	{attribute 'TcIecLibraryType'}
	{attribute 'external_name' := 'F_VN_BrightBorderObjects_GUID_85963068_12EB_DB9B_82A7_C723E1DC205C'}
	(* Find bright objects connected to the image border within a gray-scale single-channel image. *)
	FUNCTION F_VN_BrightBorderObjects : HRESULT
	VAR_INPUT
		ipSrcImage	:	ITcVnImage;	(* Source image (USINT, UINT, INT, REAL, or LREAL, 1 channel) *)
		ipDestImage	:	REFERENCE TO ITcVnImage;	(* Destination image (An appropriate destination image will be created if required.) *)
		hrPrev	:	HRESULT;	(* HRESULT indicating the result of previous operations (If SUCCEEDED(hrPrev) equals false, no operation is executed.) *)
	END_VAR

END_FUNCTION

// Functions/Image Filtering/F_VN_CreateStructuringElement

	{attribute 'TcIecLibraryType'}
	{attribute 'external_name' := 'F_VN_CreateStructuringElement_GUID_A74CE5A4_39AA_D057_BA78_297FA60F12C8'}
	(* Creates a structuring element for the usage with morphological operators and allocate an appropriate data buffer. The initial reference count is set to one if a new image interface is created and kept, otherwise. *)
	FUNCTION F_VN_CreateStructuringElement : HRESULT
	VAR_INPUT
		ipStructuringElement	:	REFERENCE TO ITcVnImage;	(* Returns the created structuring element (Non-zero interface pointers are reused.) *)
		eShape	:	ETcVnStructuringElementShape;	(* Shape of the structuring element (rectangle, cross, or ellipse) *)
		nWidth	:	UDINT;	(* Width *)
		nHeight	:	UDINT;	(* Height *)
		hrPrev	:	HRESULT;	(* HRESULT indicating the result of previous operations (If SUCCEEDED(hrPrev) equals false, no operation is executed.) *)
	END_VAR

END_FUNCTION

// Functions/Image Filtering/F_VN_CustomFilter

	{attribute 'TcIecLibraryType'}
	{attribute 'external_name' := 'F_VN_CustomFilter_GUID_4301F747_474B_D00C_9989_9E35727DC697'}
	(* Apply a custom filter to the image. *)
	FUNCTION F_VN_CustomFilter : HRESULT
	VAR_INPUT
		ipSrcImage	:	ITcVnImage;	(* Source image *)
		ipDestImage	:	REFERENCE TO ITcVnImage;	(* Destination image (An appropriate destination image will be created if required.) *)
		eDestDepth	:	ETcVnElementType;	(* Destination image depth *)
	END_VAR
	VAR_IN_OUT
		stKernel	:	TcVnMatrix;	(* Custom filter kernel with values of type REAL or LREAL *)
	END_VAR
	VAR_INPUT
		hrPrev	:	HRESULT;	(* HRESULT indicating the result of previous operations (If SUCCEEDED(hrPrev) equals false, no operation is executed.) *)
	END_VAR

END_FUNCTION

// Functions/Image Filtering/F_VN_CustomFilterExp

	{attribute 'TcIecLibraryType'}
	{attribute 'external_name' := 'F_VN_CustomFilterExp_GUID_6B16FEA9_6021_D269_AEDC_2F022CED5005'}
	(* Apply a custom filter to the image. (expert function) *)
	FUNCTION F_VN_CustomFilterExp : HRESULT
	VAR_INPUT
		ipSrcImage	:	ITcVnImage;	(* Source image *)
		ipDestImage	:	REFERENCE TO ITcVnImage;	(* Destination image (An appropriate destination image will be created if required.) *)
		eDestDepth	:	ETcVnElementType;	(* Destination image depth *)
	END_VAR
	VAR_IN_OUT
		stKernel	:	TcVnMatrix;	(* Custom filter kernel with values of type REAL or LREAL *)
		aAnchor	:	TcVnPoint;	(* Anchor point of the kernel *)
	END_VAR
	VAR_INPUT
		fDelta	:	LREAL;	(* Value added to each pixel after filtering *)
		eBorderType	:	ETcVnBorderInterpolationMethod;	(* Image border handling *)
		hrPrev	:	HRESULT;	(* HRESULT indicating the result of previous operations (If SUCCEEDED(hrPrev) equals false, no operation is executed.) *)
	END_VAR

END_FUNCTION

// Functions/Image Filtering/F_VN_DarkBorderObjects

	{attribute 'TcIecLibraryType'}
	{attribute 'external_name' := 'F_VN_DarkBorderObjects_GUID_502A5401_CBE1_DB60_8EE9_DC582F5D3E12'}
	(* Find dark objects connected to the image border within a gray-scale single-channel image. (equivalent to filling holes) *)
	FUNCTION F_VN_DarkBorderObjects : HRESULT
	VAR_INPUT
		ipSrcImage	:	ITcVnImage;	(* Source image (USINT, UINT, INT, REAL, or LREAL, 1 channel) *)
		ipDestImage	:	REFERENCE TO ITcVnImage;	(* Destination image (An appropriate destination image will be created if required.) *)
		hrPrev	:	HRESULT;	(* HRESULT indicating the result of previous operations (If SUCCEEDED(hrPrev) equals false, no operation is executed.) *)
	END_VAR

END_FUNCTION

// Functions/Image Filtering/F_VN_FillHoles

	{attribute 'TcIecLibraryType'}
	{attribute 'external_name' := 'F_VN_FillHoles_GUID_355DF251_1290_D7ED_B630_2E4E8A66643C'}
	(* Fill holes within a gray-scale single-channel image. (equivalent to finding dark border objects) *)
	FUNCTION F_VN_FillHoles : HRESULT
	VAR_INPUT
		ipSrcImage	:	ITcVnImage;	(* Source image (USINT, UINT, INT, REAL, or LREAL, 1 channel) *)
		ipDestImage	:	REFERENCE TO ITcVnImage;	(* Destination image (An appropriate destination image will be created if required.) *)
		hrPrev	:	HRESULT;	(* HRESULT indicating the result of previous operations (If SUCCEEDED(hrPrev) equals false, no operation is executed.) *)
	END_VAR

END_FUNCTION

// Functions/Image Filtering/F_VN_GaussianFilter

	{attribute 'TcIecLibraryType'}
	{attribute 'external_name' := 'F_VN_GaussianFilter_GUID_E5394B01_3A0E_DAE0_9B18_9A4594D869A5'}
	(* Apply a Gaussian filter to smooth the image. *)
	FUNCTION F_VN_GaussianFilter : HRESULT
	VAR_INPUT
		ipSrcImage	:	ITcVnImage;	(* Source image *)
		ipDestImage	:	REFERENCE TO ITcVnImage;	(* Destination image (An appropriate destination image will be created if required.) *)
		nFilterWidth	:	UDINT;	(* Filter width in pixels (1, 3, 5, 7, ...) *)
		nFilterHeight	:	UDINT;	(* Filter height in pixels (1, 3, 5, 7, ...) *)
		hrPrev	:	HRESULT;	(* HRESULT indicating the result of previous operations (If SUCCEEDED(hrPrev) equals false, no operation is executed.) *)
	END_VAR

END_FUNCTION

// Functions/Image Filtering/F_VN_GaussianFilterExp

	{attribute 'TcIecLibraryType'}
	{attribute 'external_name' := 'F_VN_GaussianFilterExp_GUID_34305DF4_4689_DEA9_9855_ED8AC64FC35B'}
	(* Apply a Gaussian filter to smooth the image. (expert function) *)
	FUNCTION F_VN_GaussianFilterExp : HRESULT
	VAR_INPUT
		ipSrcImage	:	ITcVnImage;	(* Source image *)
		ipDestImage	:	REFERENCE TO ITcVnImage;	(* Destination image (An appropriate destination image will be created if required.) *)
		nFilterWidth	:	UDINT;	(* Filter width in pixels (1, 3, 5, 7, ...) *)
		nFilterHeight	:	UDINT;	(* Filter height in pixels (1, 3, 5, 7, ...) *)
		fSigmaX	:	LREAL;	(* Gaussian kernel standard deviation in X direction (>= 0, automatically chosen if 0) *)
		fSigmaY	:	LREAL;	(* Gaussian kernel standard deviation in Y direction (>= 0, automatically chosen if 0) *)
		eBorderType	:	ETcVnBorderInterpolationMethod;	(* Image border handling *)
		hrPrev	:	HRESULT;	(* HRESULT indicating the result of previous operations (If SUCCEEDED(hrPrev) equals false, no operation is executed.) *)
	END_VAR

END_FUNCTION

// Functions/Image Filtering/F_VN_LaplacianFilter

	{attribute 'TcIecLibraryType'}
	{attribute 'external_name' := 'F_VN_LaplacianFilter_GUID_52689B07_71D3_DE56_A0C0_525AA2EFFA66'}
	(* Apply a Laplacian filter to an image. *)
	FUNCTION F_VN_LaplacianFilter : HRESULT
	VAR_INPUT
		ipSrcImage	:	ITcVnImage;	(* Source image *)
		ipDestImage	:	REFERENCE TO ITcVnImage;	(* Destination image (An appropriate destination image will be created if required.) *)
		eDestDepth	:	ETcVnElementType;	(* Destination image depth *)
		hrPrev	:	HRESULT;	(* HRESULT indicating the result of previous operations (If SUCCEEDED(hrPrev) equals false, no operation is executed.) *)
	END_VAR

END_FUNCTION

// Functions/Image Filtering/F_VN_LaplacianFilterExp

	{attribute 'TcIecLibraryType'}
	{attribute 'external_name' := 'F_VN_LaplacianFilterExp_GUID_F05E54BA_3338_DB0A_A7D6_DE17DEB649CB'}
	(* Apply a Laplacian filter to an image. (expert function) *)
	FUNCTION F_VN_LaplacianFilterExp : HRESULT
	VAR_INPUT
		ipSrcImage	:	ITcVnImage;	(* Source image *)
		ipDestImage	:	REFERENCE TO ITcVnImage;	(* Destination image (An appropriate destination image will be created if required.) *)
		eDestDepth	:	ETcVnElementType;	(* Destination image depth *)
		nKernelSize	:	UDINT;	(* Aperture size used to compute the second-derivative filters (1, 3, 5, ..., 31) *)
		fScale	:	LREAL;	(* Scale factor for the computed derivative values *)
		fDelta	:	LREAL;	(* Delta value that is added to the results before storing them *)
		eBorderType	:	ETcVnBorderInterpolationMethod;	(* Image border handling *)
		hrPrev	:	HRESULT;	(* HRESULT indicating the result of previous operations (If SUCCEEDED(hrPrev) equals false, no operation is executed.) *)
	END_VAR

END_FUNCTION

// Functions/Image Filtering/F_VN_LocalMaxima

	{attribute 'TcIecLibraryType'}
	{attribute 'external_name' := 'F_VN_LocalMaxima_GUID_73E2BFA3_7B8C_D368_9D3A_ABFF9FB011DB'}
	(* Find local maxima in a gray-scale single-channel image. The found maxima are marked by a value of 1 in the destination image. *)
	FUNCTION F_VN_LocalMaxima : HRESULT
	VAR_INPUT
		ipSrcImage	:	ITcVnImage;	(* Source image (USINT or UINT, 1 channel) *)
		ipDestImage	:	REFERENCE TO ITcVnImage;	(* Destination image (Must be different from ipSrcImage! An appropriate destination image will be created if required.) *)
		hrPrev	:	HRESULT;	(* HRESULT indicating the result of previous operations (If SUCCEEDED(hrPrev) equals false, no operation is executed.) *)
	END_VAR

END_FUNCTION

// Functions/Image Filtering/F_VN_LocalMinima

	{attribute 'TcIecLibraryType'}
	{attribute 'external_name' := 'F_VN_LocalMinima_GUID_43B2D13E_E00E_D8F8_8DF7_26EA4EF5D134'}
	(* Find local minima in a gray-scale single-channel image. The found minima are marked by a value of 1 in the destination image. *)
	FUNCTION F_VN_LocalMinima : HRESULT
	VAR_INPUT
		ipSrcImage	:	ITcVnImage;	(* Source image (USINT or UINT, 1 channel) *)
		ipDestImage	:	REFERENCE TO ITcVnImage;	(* Destination image (Must be different from ipSrcImage! An appropriate destination image will be created if required.) *)
		hrPrev	:	HRESULT;	(* HRESULT indicating the result of previous operations (If SUCCEEDED(hrPrev) equals false, no operation is executed.) *)
	END_VAR

END_FUNCTION

// Functions/Image Filtering/F_VN_MedianFilter

	{attribute 'TcIecLibraryType'}
	{attribute 'external_name' := 'F_VN_MedianFilter_GUID_68A1C045_786D_D318_9650_B93B817DB87C'}
	(* Apply a Median filter to an image. *)
	FUNCTION F_VN_MedianFilter : HRESULT
	VAR_INPUT
		ipSrcImage	:	ITcVnImage;	(* Source image (for nFilterSize 3 or 5: USINT, UINT, REAL. For bigger filters, only USINT is supported. *)
		ipDestImage	:	REFERENCE TO ITcVnImage;	(* Destination image (An appropriate destination image will be created if required.) *)
		nFilterSize	:	UDINT;	(* Size (width and height) of the filter (3, 5, 7, ...) *)
		hrPrev	:	HRESULT;	(* HRESULT indicating the result of previous operations (If SUCCEEDED(hrPrev) equals false, no operation is executed.) *)
	END_VAR

END_FUNCTION

// Functions/Image Filtering/F_VN_MorphologicalOperator

	{attribute 'TcIecLibraryType'}
	{attribute 'external_name' := 'F_VN_MorphologicalOperator_GUID_C2AADC35_1A3C_DECA_BADD_187CC41E0AFB'}
	(* Apply a morphological operator. *)
	FUNCTION F_VN_MorphologicalOperator : HRESULT
	VAR_INPUT
		ipSrcImage	:	ITcVnImage;	(* Source image (only 1 channel supported for reconstruction operators) *)
		ipDestImage	:	REFERENCE TO ITcVnImage;	(* Destination image (An appropriate destination image will be created if required.) *)
		eOperator	:	ETcVnMorphologicalOperator;	(* Operator type *)
		ipStructuringElement	:	ITcVnImage;	(* Structuring element to be applied (Typically created via F_VN_CreateStructuringElement.) *)
		hrPrev	:	HRESULT;	(* HRESULT indicating the result of previous operations (If SUCCEEDED(hrPrev) equals false, no operation is executed.) *)
	END_VAR

END_FUNCTION

// Functions/Image Filtering/F_VN_RemoveLocalMaxima

	{attribute 'TcIecLibraryType'}
	{attribute 'external_name' := 'F_VN_RemoveLocalMaxima_GUID_133B4553_4F99_DBCD_BA62_EA37E8765D5B'}
	(* Remove local maxima up to a given height from a gray-scale single-channel image. *)
	FUNCTION F_VN_RemoveLocalMaxima : HRESULT
	VAR_INPUT
		ipSrcImage	:	ITcVnImage;	(* Source image (USINT, UINT, INT, REAL, or LREAL, 1 channel) *)
		ipDestImage	:	REFERENCE TO ITcVnImage;	(* Destination image (An appropriate destination image will be created if required.) *)
		fHeight	:	LREAL;	(* Maximum height of the maxima to be removed (must be greater than 0) *)
		hrPrev	:	HRESULT;	(* HRESULT indicating the result of previous operations (If SUCCEEDED(hrPrev) equals false, no operation is executed.) *)
	END_VAR

END_FUNCTION

// Functions/Image Filtering/F_VN_RemoveLocalMinima

	{attribute 'TcIecLibraryType'}
	{attribute 'external_name' := 'F_VN_RemoveLocalMinima_GUID_A59442F0_2AE9_D045_8F9C_09A3C82C0A3B'}
	(* Remove local minima up to a given height from a gray-scale single-channel image. *)
	FUNCTION F_VN_RemoveLocalMinima : HRESULT
	VAR_INPUT
		ipSrcImage	:	ITcVnImage;	(* Source image (USINT, UINT, INT, REAL, or LREAL, 1 channel) *)
		ipDestImage	:	REFERENCE TO ITcVnImage;	(* Destination image (An appropriate destination image will be created if required.) *)
		fHeight	:	LREAL;	(* Maximum height of the minima to be removed (must be greater than 0) *)
		hrPrev	:	HRESULT;	(* HRESULT indicating the result of previous operations (If SUCCEEDED(hrPrev) equals false, no operation is executed.) *)
	END_VAR

END_FUNCTION

// Functions/Image Filtering/F_VN_ScharrFilter

	{attribute 'TcIecLibraryType'}
	{attribute 'external_name' := 'F_VN_ScharrFilter_GUID_3CD4A752_576C_D682_949F_3ED3E34C66A7'}
	(* Calculates the first order derivative in x or y direction using a Scharr filter. *)
	FUNCTION F_VN_ScharrFilter : HRESULT
	VAR_INPUT
		ipSrcImage	:	ITcVnImage;	(* Source image *)
		ipDestImage	:	REFERENCE TO ITcVnImage;	(* Destination image (An appropriate destination image will be created if required.) *)
		eDestDepth	:	ETcVnElementType;	(* Destination image depth *)
		eFilterDirection	:	ETcVnFilterDirection;	(* Filter direction *)
		hrPrev	:	HRESULT;	(* HRESULT indicating the result of previous operations (If SUCCEEDED(hrPrev) equals false, no operation is executed.) *)
	END_VAR

END_FUNCTION

// Functions/Image Filtering/F_VN_ScharrFilterExp

	{attribute 'TcIecLibraryType'}
	{attribute 'external_name' := 'F_VN_ScharrFilterExp_GUID_14964554_311A_DD6B_9094_26927304E48F'}
	(* Calculates the first order derivative in x or y direction using a Scharr filter. (expert function) *)
	FUNCTION F_VN_ScharrFilterExp : HRESULT
	VAR_INPUT
		ipSrcImage	:	ITcVnImage;	(* Source image *)
		ipDestImage	:	REFERENCE TO ITcVnImage;	(* Destination image (An appropriate destination image will be created if required.) *)
		eDestDepth	:	ETcVnElementType;	(* Destination image depth *)
		eFilterDirection	:	ETcVnFilterDirection;	(* Filter direction *)
		fScale	:	LREAL;	(* Scale factor for the computed derivative values *)
		fDelta	:	LREAL;	(* Delta value that is added to the results prior to storing them in dest *)
		eBorderType	:	ETcVnBorderInterpolationMethod;	(* Image border handling *)
		hrPrev	:	HRESULT;	(* HRESULT indicating the result of previous operations (If SUCCEEDED(hrPrev) equals false, no operation is executed.) *)
	END_VAR

END_FUNCTION

// Functions/Image Filtering/F_VN_SeparableCustomFilter

	{attribute 'TcIecLibraryType'}
	{attribute 'external_name' := 'F_VN_SeparableCustomFilter_GUID_638E373F_2CCD_D425_B656_29701E8F04DD'}
	(* Apply a separable custom filter to the image. *)
	FUNCTION F_VN_SeparableCustomFilter : HRESULT
	VAR_INPUT
		ipSrcImage	:	ITcVnImage;	(* Source image *)
		ipDestImage	:	REFERENCE TO ITcVnImage;	(* Destination image (An appropriate destination image will be created if required.) *)
		eDestDepth	:	ETcVnElementType;	(* Destination image depth *)
	END_VAR
	VAR_IN_OUT
		stKernelX	:	TcVnMatrix;	(* 1D custom row-filter kernel with values of type REAL or LREAL *)
		stKernelY	:	TcVnMatrix;	(* 1D custom column-filter kernel with values of type REAL or LREAL *)
	END_VAR
	VAR_INPUT
		hrPrev	:	HRESULT;	(* HRESULT indicating the result of previous operations (If SUCCEEDED(hrPrev) equals false, no operation is executed.) *)
	END_VAR

END_FUNCTION

// Functions/Image Filtering/F_VN_SeparableCustomFilterExp

	{attribute 'TcIecLibraryType'}
	{attribute 'external_name' := 'F_VN_SeparableCustomFilterExp_GUID_CC5A19A5_2D1C_D6B1_9D4E_5D5FBFBA8823'}
	(* Apply a separable custom filter to the image. (expert function) *)
	FUNCTION F_VN_SeparableCustomFilterExp : HRESULT
	VAR_INPUT
		ipSrcImage	:	ITcVnImage;	(* Source image *)
		ipDestImage	:	REFERENCE TO ITcVnImage;	(* Destination image (An appropriate destination image will be created if required.) *)
		eDestDepth	:	ETcVnElementType;	(* Destination image depth *)
	END_VAR
	VAR_IN_OUT
		stKernelX	:	TcVnMatrix;	(* 1D custom row-filter kernel with values of type REAL or LREAL *)
		stKernelY	:	TcVnMatrix;	(* 1D custom column-filter kernel with values of type REAL or LREAL *)
		aAnchor	:	TcVnPoint;	(* Anchor point of the kernel *)
	END_VAR
	VAR_INPUT
		fDelta	:	LREAL;	(* Value added to each pixel after filtering *)
		eBorderType	:	ETcVnBorderInterpolationMethod;	(* Image border handling *)
		hrPrev	:	HRESULT;	(* HRESULT indicating the result of previous operations (If SUCCEEDED(hrPrev) equals false, no operation is executed.) *)
	END_VAR

END_FUNCTION

// Functions/Image Filtering/F_VN_SobelFilter

	{attribute 'TcIecLibraryType'}
	{attribute 'external_name' := 'F_VN_SobelFilter_GUID_78B78962_D304_DC9E_9463_CADAFAF8E1E8'}
	(* Calculates the first, second, or mixed image derivatives using an extended Sobel filter. *)
	FUNCTION F_VN_SobelFilter : HRESULT
	VAR_INPUT
		ipSrcImage	:	ITcVnImage;	(* Source image *)
		ipDestImage	:	REFERENCE TO ITcVnImage;	(* Destination image (An appropriate destination image will be created if required.) *)
		eDestDepth	:	ETcVnElementType;	(* Destination image depth *)
		nXOrder	:	UDINT;	(* Order of the x-derivative (0, 1, 2) *)
		nYOrder	:	UDINT;	(* Order of the y-derivative (0, 1, 2) *)
		hrPrev	:	HRESULT;	(* HRESULT indicating the result of previous operations (If SUCCEEDED(hrPrev) equals false, no operation is executed.) *)
	END_VAR

END_FUNCTION

// Functions/Image Filtering/F_VN_SobelFilterExp

	{attribute 'TcIecLibraryType'}
	{attribute 'external_name' := 'F_VN_SobelFilterExp_GUID_FBDFA23E_B87D_D101_BF7D_FD7D1B526F5F'}
	(* Calculates the first, second, third, or mixed image derivatives using an extended Sobel filter. (expert function) *)
	FUNCTION F_VN_SobelFilterExp : HRESULT
	VAR_INPUT
		ipSrcImage	:	ITcVnImage;	(* Source image *)
		ipDestImage	:	REFERENCE TO ITcVnImage;	(* Destination image (An appropriate destination image will be created if required.) *)
		eDestDepth	:	ETcVnElementType;	(* Destination image depth *)
		nXOrder	:	UDINT;	(* Order of the x-derivative (must be < nKernelSize) *)
		nYOrder	:	UDINT;	(* Order of the y-derivative (must be < nKernelSize) *)
		nKernelSize	:	UDINT;	(* Size of the extended Sobel kernel (3, 5, 7, ..., 31) *)
		fScale	:	LREAL;	(* Scale factor for the computed derivative values *)
		fDelta	:	LREAL;	(* Delta value that is added to the results prior to storing them in dest *)
		eBorderType	:	ETcVnBorderInterpolationMethod;	(* Image border handling *)
		hrPrev	:	HRESULT;	(* HRESULT indicating the result of previous operations (If SUCCEEDED(hrPrev) equals false, no operation is executed.) *)
	END_VAR

END_FUNCTION

// Functions/Image Filtering/F_VN_VarianceFilter

	{attribute 'TcIecLibraryType'}
	{attribute 'external_name' := 'F_VN_VarianceFilter_GUID_725DC025_4725_DBB8_87EE_9B5A9A457993'}
	(* Calculates the local variance of an image. *)
	FUNCTION F_VN_VarianceFilter : HRESULT
	VAR_INPUT
		ipSrcImage	:	ITcVnImage;	(* Source image. Only TCVN_ET_USINT Type is supported.  *)
		ipDestImage	:	REFERENCE TO ITcVnImage;	(* Destination image of type TCVN_ET_UINT (An appropriate destination image will be created if required.) *)
		nKernelSize	:	UDINT;	(* Size of the kernel *)
		hrPrev	:	HRESULT;	(* HRESULT indicating the result of previous operations (If SUCCEEDED(hrPrev) equals false, no operation is executed.) *)
	END_VAR

END_FUNCTION

// Functions/Image Filtering/F_VN_VarianceFilterExp

	{attribute 'TcIecLibraryType'}
	{attribute 'external_name' := 'F_VN_VarianceFilterExp_GUID_3855C0A3_9566_D39D_A345_6FBD0245882C'}
	(* Calculates the local variance of an image. (expert function) *)
	FUNCTION F_VN_VarianceFilterExp : HRESULT
	VAR_INPUT
		ipSrcImage	:	ITcVnImage;	(* Source image. Only TCVN_ET_USINT Type is supported. *)
		ipDestImage	:	REFERENCE TO ITcVnImage;	(* Destination image of type TCVN_ET_UINT (An appropriate destination image will be created if required.) *)
		nKernelSize	:	UDINT;	(* Size of the kernel *)
		fScale	:	LREAL;	(* Scale factor for the computed variance values *)
		eBorderType	:	ETcVnBorderInterpolationMethod;	(* Image border handling *)
		hrPrev	:	HRESULT;	(* HRESULT indicating the result of previous operations (If SUCCEEDED(hrPrev) equals false, no operation is executed.) *)
	END_VAR

END_FUNCTION

// Functions/Miscellaneous/F_VN_CheckFunctionInitialization

	{attribute 'TcIecLibraryType'}
	{attribute 'external_name' := 'F_VN_CheckFunctionInitialization_GUID_5C1CCB2A_8EAF_D10A_81E3_298A44F01F89'}
	(* Check if a function is initialized with the specified options. *)
	FUNCTION F_VN_CheckFunctionInitialization : HRESULT
	VAR_INPUT
		eFunction	:	ETcVnInitializableFunction;	(* Initializable function *)
		nOptions	:	ULINT;	(* Initialization options for the function *)
		hrPrev	:	HRESULT;	(* HRESULT indicating the result of previous operations (If SUCCEEDED(hrPrev) equals false, no operation is executed.) *)
	END_VAR

END_FUNCTION

// Functions/Miscellaneous/F_VN_ClipLineToBoundary

	{attribute 'TcIecLibraryType'}
	{attribute 'external_name' := 'F_VN_ClipLineToBoundary_GUID_C41C5126_7C61_D48E_9219_1D6808E929F9'}
	(* Clips a line to a rectangular boundary. *)
	FUNCTION F_VN_ClipLineToBoundary : HRESULT
	VAR_IN_OUT
		aLine	:	TcVnVector4_LREAL;	(* The first and second element describe the x and y component of the direction vector. The third and fourth element describe the x and y component of the position vector. *)
	END_VAR
	VAR_INPUT
		nX1	:	DINT;	(* x of top left rectangle point *)
		nY1	:	DINT;	(* y of top left rectangle point *)
		nX2	:	DINT;	(* x of bottom right rectangle point *)
		nY2	:	DINT;	(* Y of bottom right rectangle point *)
	END_VAR
	VAR_IN_OUT
		aStartPoint	:	TcVnPoint2_REAL;	(* Returns the clipped starting point of the line. *)
		aEndPoint	:	TcVnPoint2_REAL;	(* Returns the clipped end point of the line. *)
	END_VAR
	VAR_INPUT
		hrPrev	:	HRESULT;	(* HRESULT indicating the result of previous operations (If SUCCEEDED(hrPrev) equals false, no operation is executed.) *)
	END_VAR

END_FUNCTION

// Functions/Miscellaneous/F_VN_ClipLineToBoundary_ITcVnImage

	{attribute 'TcIecLibraryType'}
	{attribute 'external_name' := 'F_VN_ClipLineToBoundary_ITcVnImage_GUID_7F54C3D6_7EC7_D30D_888C_AFEC76DB700F'}
	(* Clips a line to the boundary of an image. *)
	FUNCTION F_VN_ClipLineToBoundary_ITcVnImage : HRESULT
	VAR_IN_OUT
		aLine	:	TcVnVector4_LREAL;	(* The first and second element describe the x and y component of the direction vector. The third and fourth element describe the x and y component of the position vector. *)
	END_VAR
	VAR_INPUT
		ipImage	:	ITcVnImage;	(* Image, from which to derive the boundary *)
	END_VAR
	VAR_IN_OUT
		aStartPoint	:	TcVnPoint2_REAL;	(* Returns the clipped starting point of the line. *)
		aEndPoint	:	TcVnPoint2_REAL;	(* Returns the clipped end point of the line. *)
	END_VAR
	VAR_INPUT
		hrPrev	:	HRESULT;	(* HRESULT indicating the result of previous operations (If SUCCEEDED(hrPrev) equals false, no operation is executed.) *)
	END_VAR

END_FUNCTION

// Functions/Miscellaneous/F_VN_ClipLineToBoundary_TcVnRectangle_DINT

	{attribute 'TcIecLibraryType'}
	{attribute 'external_name' := 'F_VN_ClipLineToBoundary_TcVnRectangle_DINT_GUID_1C947EAF_E2B4_D27E_9C79_9E84C29C006C'}
	(* Clips a line to a rectangular boundary. *)
	FUNCTION F_VN_ClipLineToBoundary_TcVnRectangle_DINT : HRESULT
	VAR_IN_OUT
		aLine	:	TcVnVector4_LREAL;	(* The first and second element describe the x and y component of the direction vector. The third and fourth element describe the x and y component of the position vector. *)
		stRectangle	:	TcVnRectangle_DINT;	(* Rectangular boundary *)
		aStartPoint	:	TcVnPoint2_REAL;	(* Returns the clipped starting point of the line. *)
		aEndPoint	:	TcVnPoint2_REAL;	(* Returns the clipped end point of the line. *)
	END_VAR
	VAR_INPUT
		hrPrev	:	HRESULT;	(* HRESULT indicating the result of previous operations (If SUCCEEDED(hrPrev) equals false, no operation is executed.) *)
	END_VAR

END_FUNCTION

// Functions/Miscellaneous/F_VN_ConvertITcUnknownToITcVnBitmapExport

	{attribute 'TcIecLibraryType'}
	{attribute 'external_name' := 'F_VN_ConvertITcUnknownToITcVnBitmapExport_GUID_B532B9D8_E0C1_D2FB_8DFC_5214526A5A63'}
	(* Convert an ITcUnknown interface pointer to an ITcVnBitmapExport interface pointer. The destination pointer will be released (if existing) and set to the source pointer. The source pointer will be set to 0. *)
	FUNCTION F_VN_ConvertITcUnknownToITcVnBitmapExport : HRESULT
	VAR_INPUT
		ipSrc	:	REFERENCE TO ITcUnknown;	(* Source pointer *)
		ipDest	:	REFERENCE TO ITcVnBitmapExport;	(* Destination pointer *)
		hrPrev	:	HRESULT;	(* HRESULT indicating the result of previous operations (If SUCCEEDED(hrPrev) equals false, no operation is executed.) *)
	END_VAR

END_FUNCTION

// Functions/Miscellaneous/F_VN_ConvertITcUnknownToITcVnContainer

	{attribute 'TcIecLibraryType'}
	{attribute 'external_name' := 'F_VN_ConvertITcUnknownToITcVnContainer_GUID_880EE029_87B5_D470_B6E3_1020C4DE5402'}
	(* Convert an ITcUnknown interface pointer to an ITcVnContainer interface pointer. The destination pointer will be released (if existing) and set to the source pointer. The source pointer will be set to 0. *)
	FUNCTION F_VN_ConvertITcUnknownToITcVnContainer : HRESULT
	VAR_INPUT
		ipSrc	:	REFERENCE TO ITcUnknown;	(* Source pointer *)
		ipDest	:	REFERENCE TO ITcVnContainer;	(* Destination pointer *)
		hrPrev	:	HRESULT;	(* HRESULT indicating the result of previous operations (If SUCCEEDED(hrPrev) equals false, no operation is executed.) *)
	END_VAR

END_FUNCTION

// Functions/Miscellaneous/F_VN_ConvertITcUnknownToITcVnImage

	{attribute 'TcIecLibraryType'}
	{attribute 'external_name' := 'F_VN_ConvertITcUnknownToITcVnImage_GUID_87F6AF06_A93F_DC2A_9949_25D97D734767'}
	(* Convert an ITcUnknown interface pointer to an ITcVnImage interface pointer. The destination pointer will be released (if existing) and set to the source pointer. The source pointer will be set to 0. *)
	FUNCTION F_VN_ConvertITcUnknownToITcVnImage : HRESULT
	VAR_INPUT
		ipSrc	:	REFERENCE TO ITcUnknown;	(* Source pointer *)
		ipDest	:	REFERENCE TO ITcVnImage;	(* Destination pointer *)
		hrPrev	:	HRESULT;	(* HRESULT indicating the result of previous operations (If SUCCEEDED(hrPrev) equals false, no operation is executed.) *)
	END_VAR

END_FUNCTION

// Functions/Miscellaneous/F_VN_ConvertITcUnknownToITcVnMlModel

	{attribute 'TcIecLibraryType'}
	{attribute 'external_name' := 'F_VN_ConvertITcUnknownToITcVnMlModel_GUID_9B78767C_E4B6_DA9B_88E4_A7BD10FC7F72'}
	(* Convert an ITcUnknown interface pointer to an ITcVnMlModel interface pointer. The destination pointer will be released (if existing) and set to the source pointer. The source pointer will be set to 0. *)
	FUNCTION F_VN_ConvertITcUnknownToITcVnMlModel : HRESULT
	VAR_INPUT
		ipSrc	:	REFERENCE TO ITcUnknown;	(* Source pointer *)
		ipDest	:	REFERENCE TO ITcVnMlModel;	(* Destination pointer *)
		hrPrev	:	HRESULT;	(* HRESULT indicating the result of previous operations (If SUCCEEDED(hrPrev) equals false, no operation is executed.) *)
	END_VAR

END_FUNCTION

// Functions/Miscellaneous/F_VN_DeinitializeFunction

	{attribute 'TcIecLibraryType'}
	{attribute 'external_name' := 'F_VN_DeinitializeFunction_GUID_A16DDE96_C780_D4ED_B159_57D03517C793'}
	(* Deinitialize the specified options for the function. *)
	FUNCTION F_VN_DeinitializeFunction : HRESULT
	VAR_INPUT
		eFunction	:	ETcVnInitializableFunction;	(* Initializable function *)
		nOptions	:	ULINT;	(* Initialization options for the function *)
		hrPrev	:	HRESULT;	(* HRESULT indicating the result of previous operations (If SUCCEEDED(hrPrev) equals false, no operation is executed.) *)
	END_VAR

END_FUNCTION

// Functions/Miscellaneous/F_VN_GetTimestamp

	{attribute 'TcIecLibraryType'}
	{attribute 'external_name' := 'F_VN_GetTimestamp_GUID_5DF60E92_4ED1_D095_AABF_9A14F3701D57'}
	(* Get the timestamp (actual DC time) from the last change of an object (e.g. ITcVnImage or ITcVnContainer) *)
	FUNCTION F_VN_GetTimestamp : HRESULT
	VAR_INPUT
		ipUnknown	:	ITcUnknown;	(* An object implementing ITcUnknown and ITcVnTimestamp (e.g. ITcVnImage or ITcVnContainer) *)
	END_VAR
	VAR_IN_OUT
		nTimestamp	:	LINT;	(* Returns the timestamp *)
	END_VAR
	VAR_INPUT
		hrPrev	:	HRESULT;	(* HRESULT indicating the result of previous operations (If SUCCEEDED(hrPrev) equals false, no operation is executed.) *)
	END_VAR

END_FUNCTION

// Functions/Miscellaneous/F_VN_HuMomentInvariants

	{attribute 'TcIecLibraryType'}
	{attribute 'external_name' := 'F_VN_HuMomentInvariants_GUID_2711399A_D495_DC65_AA2B_5CE1A04EE2AF'}
	(* Computes the Hu moment invariants. *)
	FUNCTION F_VN_HuMomentInvariants : HRESULT
	VAR_IN_OUT
		stMoments	:	TcVnMoments;	(* Moments from which to compute the Hu invariants *)
		aHuInvariants	:	TcVnArray7_LREAL;	(* Returns the Hu moment invariants *)
	END_VAR
	VAR_INPUT
		hrPrev	:	HRESULT;	(* HRESULT indicating the result of previous operations (If SUCCEEDED(hrPrev) equals false, no operation is executed.) *)
	END_VAR

END_FUNCTION

// Functions/Miscellaneous/F_VN_InitMatrixStruct

	{attribute 'TcIecLibraryType'}
	{attribute 'external_name' := 'F_VN_InitMatrixStruct_GUID_1C09F9C6_E010_DD28_ADEA_6854B0A7D205'}
	(* Initialize a struct of the type TcVnMatrix extending a buffer with metainformation so that it can be used as a matrix. *)
	FUNCTION F_VN_InitMatrixStruct : HRESULT
	VAR_INPUT
		pSrcBuffer	:	PVOID;	(* Source buffer *)
	END_VAR
	VAR_IN_OUT
		stDestMatrix	:	TcVnMatrix;	(* Returns completed matrix struct *)
	END_VAR
	VAR_INPUT
		nRows	:	UDINT;	(* Matrix rows *)
		nCols	:	UDINT;	(* Matrix columns *)
		eElementType	:	ETcVnElementType;	(* Type of the matrix elements *)
		hrPrev	:	HRESULT;	(* HRESULT indicating the result of previous operations (If SUCCEEDED(hrPrev) equals false, no operation is executed.) *)
	END_VAR

END_FUNCTION

// Functions/Miscellaneous/F_VN_InvertMatrix3x3

	{attribute 'TcIecLibraryType'}
	{attribute 'external_name' := 'F_VN_InvertMatrix3x3_GUID_7330F74D_D9F2_DA11_9565_C54FAB9872E4'}
	(* Invert a 3x3 matrix. *)
	FUNCTION F_VN_InvertMatrix3x3 : HRESULT
	VAR_IN_OUT
		aSrcMatrix	:	TcVnMatrix3x3_LREAL;	(* Source matrix *)
		aInvertedMatrix	:	TcVnMatrix3x3_LREAL;	(* Returns inverted matrix *)
	END_VAR
	VAR_INPUT
		hrPrev	:	HRESULT;	(* HRESULT indicating the result of previous operations (If SUCCEEDED(hrPrev) equals false, no operation is executed.) *)
	END_VAR

END_FUNCTION

// Functions/Miscellaneous/F_VN_LineIntersectionPoint

	{attribute 'TcIecLibraryType'}
	{attribute 'external_name' := 'F_VN_LineIntersectionPoint_GUID_925F5E97_FC06_D9E2_A2C2_EF91F0F3DF91'}
	(* Computes the intersection point between two lines (returns S_FALSE if the provided lines are parallel). *)
	FUNCTION F_VN_LineIntersectionPoint : HRESULT
	VAR_IN_OUT
		aLine1	:	TcVnVector4_LREAL;	(* First line. The first and second element describe the x and y component of a vector collinear to the line. The third and fourth element describe the x and y component of a point on the line. *)
		aLine2	:	TcVnVector4_LREAL;	(* Second line. The first and second element describe the x and y component of a vector collinear to the line. The third and fourth element describe the x and y component of a point on the line. *)
		aIntersecPoint	:	TcVnPoint2_REAL;	(* Returns the intersection point of aLine1 and aLine2. *)
	END_VAR
	VAR_INPUT
		hrPrev	:	HRESULT;	(* HRESULT indicating the result of previous operations (If SUCCEEDED(hrPrev) equals false, no operation is executed.) *)
	END_VAR

END_FUNCTION

// Functions/Miscellaneous/F_VN_LineIntersectionPointAndAngle

	{attribute 'TcIecLibraryType'}
	{attribute 'external_name' := 'F_VN_LineIntersectionPointAndAngle_GUID_992DA0B1_86B9_D837_A5E3_111787A70BA8'}
	(* Computes the intersection point and angle between two lines (returns S_FALSE if the provided lines are parallel). *)
	FUNCTION F_VN_LineIntersectionPointAndAngle : HRESULT
	VAR_IN_OUT
		aLine1	:	TcVnVector4_LREAL;	(* First line. The first and second element describe the x and y component of a vector collinear to the line. The third and fourth element describe the x and y component of a point on the line. *)
		aLine2	:	TcVnVector4_LREAL;	(* Second line. The first and second element describe the x and y component of a vector collinear to the line. The third and fourth element describe the x and y component of a point on the line. *)
		aIntersecPoint	:	TcVnPoint2_REAL;	(* Returns the intersection point of aLine1 and aLine2. *)
		fAngle	:	REAL;	(* Returns the intersection angle of aLine1 and aLine2. *)
	END_VAR
	VAR_INPUT
		bAngleInDegrees	:	BOOL;	(* If TRUE, fAngle is in degrees. If FALSE, fAngle is in radians. *)
		hrPrev	:	HRESULT;	(* HRESULT indicating the result of previous operations (If SUCCEEDED(hrPrev) equals false, no operation is executed.) *)
	END_VAR

END_FUNCTION

// Functions/Miscellaneous/F_VN_MultiplyMatrices

	{attribute 'TcIecLibraryType'}
	{attribute 'external_name' := 'F_VN_MultiplyMatrices_GUID_75DAA14E_E989_DA2E_A1B5_CFD09EDDB32D'}
	(* Matrix multiplication of two matrices (A * B = C). All matrices are represented by structs holding a pointer to an array of the appropriate size. *)
	FUNCTION F_VN_MultiplyMatrices : HRESULT
	VAR_IN_OUT
		stSrcMatrix1	:	TcVnMatrix;	(* First source matrix (A) *)
		stSrcMatrix2	:	TcVnMatrix;	(* Second source matrix (B) *)
		stDestMatrix	:	TcVnMatrix;	(* Destination matrix (C) (The destination matrix is filled by this function, but the required memory needs to be provided.) *)
	END_VAR
	VAR_INPUT
		hrPrev	:	HRESULT;	(* HRESULT indicating the result of previous operations (If SUCCEEDED(hrPrev) equals false, no operation is executed.) *)
	END_VAR

END_FUNCTION

// Functions/Miscellaneous/F_VN_OrthogonalVector_TcVnVector2_DINT

	{attribute 'TcIecLibraryType'}
	{attribute 'external_name' := 'F_VN_OrthogonalVector_TcVnVector2_DINT_GUID_939CA6E7_9272_D5A1_BDF5_EA98139AD47F'}
	(* Computes an orthogonal vector to a given source vector. *)
	FUNCTION F_VN_OrthogonalVector_TcVnVector2_DINT : HRESULT
	VAR_IN_OUT
		aSrc	:	TcVnVector2_DINT;	(* Source vector *)
		aOrthogonal	:	TcVnVector2_LREAL;	(* Returns a vector orthogonal to aSrc *)
	END_VAR
	VAR_INPUT
		bNormalize	:	BOOL;	(* If true, aOrthogonal length is normalized to 1, otherwise aOrthogonal has the same length as aSrc *)
		hrPrev	:	HRESULT;	(* HRESULT indicating the result of previous operations (If SUCCEEDED(hrPrev) equals false, no operation is executed.) *)
	END_VAR

END_FUNCTION

// Functions/Miscellaneous/F_VN_OrthogonalVector_TcVnVector2_LREAL

	{attribute 'TcIecLibraryType'}
	{attribute 'external_name' := 'F_VN_OrthogonalVector_TcVnVector2_LREAL_GUID_11246D82_3A46_DFD5_9AC5_8F1C99386F60'}
	(* Computes an orthogonal vector to a given source vector. *)
	FUNCTION F_VN_OrthogonalVector_TcVnVector2_LREAL : HRESULT
	VAR_IN_OUT
		aSrc	:	TcVnVector2_LREAL;	(* Source vector *)
		aOrthogonal	:	TcVnVector2_LREAL;	(* Returns a vector orthogonal to aSrc *)
	END_VAR
	VAR_INPUT
		bNormalize	:	BOOL;	(* If true, aOrthogonal length is normalized to 1, otherwise aOrthogonal has the same length as aSrc *)
		hrPrev	:	HRESULT;	(* HRESULT indicating the result of previous operations (If SUCCEEDED(hrPrev) equals false, no operation is executed.) *)
	END_VAR

END_FUNCTION

// Functions/Miscellaneous/F_VN_OrthogonalVector_TcVnVector2_REAL

	{attribute 'TcIecLibraryType'}
	{attribute 'external_name' := 'F_VN_OrthogonalVector_TcVnVector2_REAL_GUID_AEA64A60_14A7_D4A5_9AA1_CBA51503181E'}
	(* Computes an orthogonal vector to a given source vector. *)
	FUNCTION F_VN_OrthogonalVector_TcVnVector2_REAL : HRESULT
	VAR_IN_OUT
		aSrc	:	TcVnVector2_REAL;	(* Source vector *)
		aOrthogonal	:	TcVnVector2_REAL;	(* Returns a vector orthogonal to aSrc *)
	END_VAR
	VAR_INPUT
		bNormalize	:	BOOL;	(* If true, aOrthogonal length is normalized to 1, otherwise aOrthogonal has the same length as aSrc *)
		hrPrev	:	HRESULT;	(* HRESULT indicating the result of previous operations (If SUCCEEDED(hrPrev) equals false, no operation is executed.) *)
	END_VAR

END_FUNCTION

// Functions/Miscellaneous/F_VN_PointToLineDistance_TcVnPoint2_DINT

	{attribute 'TcIecLibraryType'}
	{attribute 'external_name' := 'F_VN_PointToLineDistance_TcVnPoint2_DINT_GUID_2871B486_30E4_DE6A_A203_A366BA57C5EF'}
	(* Computes the shortest distance between a point and a line. *)
	FUNCTION F_VN_PointToLineDistance_TcVnPoint2_DINT : HRESULT
	VAR_IN_OUT
		aPoint	:	TcVnPoint2_DINT;	(* Point *)
		aLinePoint1	:	TcVnPoint2_DINT;	(* Line Point 1 *)
		aLinePoint2	:	TcVnPoint2_DINT;	(* Line Point 2 *)
		fDistance	:	LREAL;	(* Returns the distance between the point and the line *)
	END_VAR
	VAR_INPUT
		hrPrev	:	HRESULT;	(* HRESULT indicating the result of previous operations (If SUCCEEDED(hrPrev) equals false, no operation is executed.) *)
	END_VAR

END_FUNCTION

// Functions/Miscellaneous/F_VN_PointToLineDistance_TcVnPoint2_LREAL

	{attribute 'TcIecLibraryType'}
	{attribute 'external_name' := 'F_VN_PointToLineDistance_TcVnPoint2_LREAL_GUID_54112E2B_0ED6_D633_9F0E_1A5E0E1ECECA'}
	(* Computes the shortest distance between a point and a line. *)
	FUNCTION F_VN_PointToLineDistance_TcVnPoint2_LREAL : HRESULT
	VAR_IN_OUT
		aPoint	:	TcVnPoint2_LREAL;	(* Point *)
		aLinePoint1	:	TcVnPoint2_LREAL;	(* Line Point 1 *)
		aLinePoint2	:	TcVnPoint2_LREAL;	(* Line Point 2 *)
		fDistance	:	LREAL;	(* Returns the distance between the point and the line *)
	END_VAR
	VAR_INPUT
		hrPrev	:	HRESULT;	(* HRESULT indicating the result of previous operations (If SUCCEEDED(hrPrev) equals false, no operation is executed.) *)
	END_VAR

END_FUNCTION

// Functions/Miscellaneous/F_VN_PointToLineDistance_TcVnPoint2_REAL

	{attribute 'TcIecLibraryType'}
	{attribute 'external_name' := 'F_VN_PointToLineDistance_TcVnPoint2_REAL_GUID_4C4BD9BD_C849_D351_88CA_5564D329D1AE'}
	(* Computes the shortest distance between a point and a line. *)
	FUNCTION F_VN_PointToLineDistance_TcVnPoint2_REAL : HRESULT
	VAR_IN_OUT
		aPoint	:	TcVnPoint2_REAL;	(* Point *)
		aLinePoint1	:	TcVnPoint2_REAL;	(* Line Point 1 *)
		aLinePoint2	:	TcVnPoint2_REAL;	(* Line Point 2 *)
		fDistance	:	LREAL;	(* Returns the distance between the point and the line *)
	END_VAR
	VAR_INPUT
		hrPrev	:	HRESULT;	(* HRESULT indicating the result of previous operations (If SUCCEEDED(hrPrev) equals false, no operation is executed.) *)
	END_VAR

END_FUNCTION

// Functions/Miscellaneous/F_VN_PointToPointDirection_TcVnPoint2_DINT

	{attribute 'TcIecLibraryType'}
	{attribute 'external_name' := 'F_VN_PointToPointDirection_TcVnPoint2_DINT_GUID_10D86722_9426_DA14_9196_3F90BB018FD6'}
	(* Computes the direction vector between 2 points. *)
	FUNCTION F_VN_PointToPointDirection_TcVnPoint2_DINT : HRESULT
	VAR_IN_OUT
		aPoint1	:	TcVnPoint2_DINT;	(* Point 1 *)
		aPoint2	:	TcVnPoint2_DINT;	(* Point 2 *)
		aDirection	:	TcVnVector2_LREAL;	(* Returns the direction vector from aPoint1 to aPoint2 *)
	END_VAR
	VAR_INPUT
		bNormalize	:	BOOL;	(* If true, aDirection length is normalized to 1, otherwise aDirection length is the distance between aPoint1 and aPoint2 *)
		hrPrev	:	HRESULT;	(* HRESULT indicating the result of previous operations (If SUCCEEDED(hrPrev) equals false, no operation is executed.) *)
	END_VAR

END_FUNCTION

// Functions/Miscellaneous/F_VN_PointToPointDirection_TcVnPoint2_LREAL

	{attribute 'TcIecLibraryType'}
	{attribute 'external_name' := 'F_VN_PointToPointDirection_TcVnPoint2_LREAL_GUID_C4034A07_9A76_D198_800C_4C117F51550A'}
	(* Computes the direction vector between 2 points. *)
	FUNCTION F_VN_PointToPointDirection_TcVnPoint2_LREAL : HRESULT
	VAR_IN_OUT
		aPoint1	:	TcVnPoint2_LREAL;	(* Point 1 *)
		aPoint2	:	TcVnPoint2_LREAL;	(* Point 2 *)
		aDirection	:	TcVnVector2_LREAL;	(* Returns the direction vector from aPoint1 to aPoint2 *)
	END_VAR
	VAR_INPUT
		bNormalize	:	BOOL;	(* If true, aDirection length is normalized to 1, otherwise aDirection length is the distance between aPoint1 and aPoint2 *)
		hrPrev	:	HRESULT;	(* HRESULT indicating the result of previous operations (If SUCCEEDED(hrPrev) equals false, no operation is executed.) *)
	END_VAR

END_FUNCTION

// Functions/Miscellaneous/F_VN_PointToPointDirection_TcVnPoint2_REAL

	{attribute 'TcIecLibraryType'}
	{attribute 'external_name' := 'F_VN_PointToPointDirection_TcVnPoint2_REAL_GUID_66073853_6474_D07E_A1DE_683F80E1972B'}
	(* Computes the direction vector between 2 points. *)
	FUNCTION F_VN_PointToPointDirection_TcVnPoint2_REAL : HRESULT
	VAR_IN_OUT
		aPoint1	:	TcVnPoint2_REAL;	(* Point 1 *)
		aPoint2	:	TcVnPoint2_REAL;	(* Point 2 *)
		aDirection	:	TcVnVector2_REAL;	(* Returns the direction vector from aPoint1 to aPoint2 *)
	END_VAR
	VAR_INPUT
		bNormalize	:	BOOL;	(* If true, aDirection length is normalized to 1, otherwise aDirection length is the distance between aPoint1 and aPoint2 *)
		hrPrev	:	HRESULT;	(* HRESULT indicating the result of previous operations (If SUCCEEDED(hrPrev) equals false, no operation is executed.) *)
	END_VAR

END_FUNCTION

// Functions/Miscellaneous/F_VN_PointToPointDistance_TcVnPoint2_DINT

	{attribute 'TcIecLibraryType'}
	{attribute 'external_name' := 'F_VN_PointToPointDistance_TcVnPoint2_DINT_GUID_FC1AA1B0_0D24_D0B6_9682_99218624C7C4'}
	(* Computes the distance between 2 points. *)
	FUNCTION F_VN_PointToPointDistance_TcVnPoint2_DINT : HRESULT
	VAR_IN_OUT
		aPoint1	:	TcVnPoint2_DINT;	(* Point 1 *)
		aPoint2	:	TcVnPoint2_DINT;	(* Point 2 *)
		fDistance	:	LREAL;	(* Returns the distance between the points *)
	END_VAR
	VAR_INPUT
		hrPrev	:	HRESULT;	(* HRESULT indicating the result of previous operations (If SUCCEEDED(hrPrev) equals false, no operation is executed.) *)
	END_VAR

END_FUNCTION

// Functions/Miscellaneous/F_VN_PointToPointDistance_TcVnPoint2_LREAL

	{attribute 'TcIecLibraryType'}
	{attribute 'external_name' := 'F_VN_PointToPointDistance_TcVnPoint2_LREAL_GUID_05019C96_C2B7_D901_82FD_FC72630347A3'}
	(* Computes the distance between 2 points. *)
	FUNCTION F_VN_PointToPointDistance_TcVnPoint2_LREAL : HRESULT
	VAR_IN_OUT
		aPoint1	:	TcVnPoint2_LREAL;	(* Point 1 *)
		aPoint2	:	TcVnPoint2_LREAL;	(* Point 2 *)
		fDistance	:	LREAL;	(* Returns the distance between the points *)
	END_VAR
	VAR_INPUT
		hrPrev	:	HRESULT;	(* HRESULT indicating the result of previous operations (If SUCCEEDED(hrPrev) equals false, no operation is executed.) *)
	END_VAR

END_FUNCTION

// Functions/Miscellaneous/F_VN_PointToPointDistance_TcVnPoint2_REAL

	{attribute 'TcIecLibraryType'}
	{attribute 'external_name' := 'F_VN_PointToPointDistance_TcVnPoint2_REAL_GUID_9D4F6A0F_1014_D857_9026_A3B168E76E08'}
	(* Computes the distance between 2 points. *)
	FUNCTION F_VN_PointToPointDistance_TcVnPoint2_REAL : HRESULT
	VAR_IN_OUT
		aPoint1	:	TcVnPoint2_REAL;	(* Point 1 *)
		aPoint2	:	TcVnPoint2_REAL;	(* Point 2 *)
		fDistance	:	LREAL;	(* Returns the distance between the points *)
	END_VAR
	VAR_INPUT
		hrPrev	:	HRESULT;	(* HRESULT indicating the result of previous operations (If SUCCEEDED(hrPrev) equals false, no operation is executed.) *)
	END_VAR

END_FUNCTION

// Functions/Miscellaneous/F_VN_RotatedRectangleCorners

	{attribute 'TcIecLibraryType'}
	{attribute 'external_name' := 'F_VN_RotatedRectangleCorners_GUID_A9B09F43_60E2_DAC5_BA83_3735B18B76F9'}
	(* Computes the 4 corner points of a rotated rectangle. *)
	FUNCTION F_VN_RotatedRectangleCorners : HRESULT
	VAR_IN_OUT
		stRect	:	TcVnRotatedRectangle;	(* Rotated rectangle *)
		aCorners	:	TcVnArray4_Point2_REAL;	(* Returns the 4 corner points *)
	END_VAR
	VAR_INPUT
		hrPrev	:	HRESULT;	(* HRESULT indicating the result of previous operations (If SUCCEEDED(hrPrev) equals false, no operation is executed.) *)
	END_VAR

END_FUNCTION

// Functions/Miscellaneous/F_VN_RotatedRectangleIntersection

	{attribute 'TcIecLibraryType'}
	{attribute 'external_name' := 'F_VN_RotatedRectangleIntersection_GUID_04FE00A9_4E9E_D65E_BC16_66001517E2EF'}
	(* Finds the intersection of 2 rotated rectangles. *)
	FUNCTION F_VN_RotatedRectangleIntersection : HRESULT
	VAR_IN_OUT
		stRect1	:	TcVnRotatedRectangle;	(* Rotated rectangle 1 *)
		stRect2	:	TcVnRotatedRectangle;	(* Rotated rectangle 2 *)
	END_VAR
	VAR_INPUT
		ipIntersection	:	REFERENCE TO ITcVnContainer;	(* Returns the intersection points (ContainerType_Vector_TcVnPoint2_REAL, non-zero interface pointers are reused) *)
	END_VAR
	VAR_IN_OUT
		eIntersection	:	ETcVnRectangleIntersection;	(* Returns the intersection type *)
	END_VAR
	VAR_INPUT
		hrPrev	:	HRESULT;	(* HRESULT indicating the result of previous operations (If SUCCEEDED(hrPrev) equals false, no operation is executed.) *)
	END_VAR

END_FUNCTION

// Functions/Miscellaneous/F_VN_SetRngSeed

	{attribute 'TcIecLibraryType'}
	{attribute 'external_name' := 'F_VN_SetRngSeed_GUID_120CBD1C_9752_D56D_B42B_E4DF916629CF'}
	(* Sets the internal pseudo random number generator seed (intended for testing purposes only). *)
	FUNCTION F_VN_SetRngSeed : HRESULT
	VAR_INPUT
		nSeed	:	DINT;	(* seed (0 sets the generator back to its initial state) *)
		hrPrev	:	HRESULT;	(* HRESULT indicating the result of previous operations (If SUCCEEDED(hrPrev) equals false, no operation is executed.) *)
	END_VAR

END_FUNCTION

// Functions/Miscellaneous/F_VN_UpdateTimestamp

	{attribute 'TcIecLibraryType'}
	{attribute 'external_name' := 'F_VN_UpdateTimestamp_GUID_C420B907_45BC_DA3F_85D2_A109AEA6015A'}
	(* Update the timestamp of an object to the actual DC time (e.g. ITcVnImage or ITcVnContainer) *)
	FUNCTION F_VN_UpdateTimestamp : HRESULT
	VAR_INPUT
		ipUnknown	:	ITcUnknown;	(* An object implementing ITcUnknown and ITcVnTimestamp (e.g. ITcVnImage or ITcVnContainer) *)
		hrPrev	:	HRESULT;	(* HRESULT indicating the result of previous operations (If SUCCEEDED(hrPrev) equals false, no operation is executed.) *)
	END_VAR

END_FUNCTION

// Functions/Basic Image Operations/F_VN_CombineImageChannels

	{attribute 'TcIecLibraryType'}
	{attribute 'external_name' := 'F_VN_CombineImageChannels_GUID_5544D388_E180_D600_BEC3_5C6BB1A16468'}
	(* Combines several single-channel images into one multi-channel image. *)
	FUNCTION F_VN_CombineImageChannels : HRESULT
	VAR_INPUT
		pSrcImages	:	PVOID;	(* Pointer to an array of single-channel source images *)
		ipDestImage	:	REFERENCE TO ITcVnImage;	(* Multi-channel destination image (An appropriate destination image will be created if required.) *)
		nSrcArraySize	:	UINT;	(* pSrcImages array size *)
		hrPrev	:	HRESULT;	(* HRESULT indicating the result of previous operations (If SUCCEEDED(hrPrev) equals false, no operation is executed.) *)
	END_VAR

END_FUNCTION

// Functions/Basic Image Operations/F_VN_ConvertElementType

	{attribute 'TcIecLibraryType'}
	{attribute 'external_name' := 'F_VN_ConvertElementType_GUID_F4FE286B_0EC9_DFB0_957A_06101850D40C'}
	(* Converts an image to another element type. *)
	FUNCTION F_VN_ConvertElementType : HRESULT
	VAR_INPUT
		ipSrcImage	:	ITcVnImage;	(* Source image *)
		ipDestImage	:	REFERENCE TO ITcVnImage;	(* Destination image (An appropriate destination image will be created if required.) *)
		eElementType	:	ETcVnElementType;	(* Desired element type of the destination image *)
		hrPrev	:	HRESULT;	(* HRESULT indicating the result of previous operations (If SUCCEEDED(hrPrev) equals false, no operation is executed.) *)
	END_VAR

END_FUNCTION

// Functions/Basic Image Operations/F_VN_ConvertElementTypeExp

	{attribute 'TcIecLibraryType'}
	{attribute 'external_name' := 'F_VN_ConvertElementTypeExp_GUID_0409B741_6FA5_D34D_8C63_1C125B4CC857'}
	(* Converts an image to another element type. (expert function) *)
	FUNCTION F_VN_ConvertElementTypeExp : HRESULT
	VAR_INPUT
		ipSrcImage	:	ITcVnImage;	(* Source image *)
		ipDestImage	:	REFERENCE TO ITcVnImage;	(* Destination image (An appropriate destination image will be created if required.) *)
		eElementType	:	ETcVnElementType;	(* Desired element type of the destination image *)
		fScaleFactor	:	LREAL;	(* Scale factor for the pixel values *)
		fDelta	:	LREAL;	(* Value that is added to the scaled pixel values *)
		hrPrev	:	HRESULT;	(* HRESULT indicating the result of previous operations (If SUCCEEDED(hrPrev) equals false, no operation is executed.) *)
	END_VAR

END_FUNCTION

// Functions/Basic Image Operations/F_VN_CopyImage

	{attribute 'TcIecLibraryType'}
	{attribute 'external_name' := 'F_VN_CopyImage_GUID_AA51C43A_5970_D6C2_A6B2_7BA7E795DF94'}
	(* Creates a deep copy of an image. *)
	FUNCTION F_VN_CopyImage : HRESULT
	VAR_INPUT
		ipSrcImage	:	ITcVnImage;	(* Source image *)
		ipDestImage	:	REFERENCE TO ITcVnImage;	(* Destination image (An appropriate destination image will be created if required.) *)
		hrPrev	:	HRESULT;	(* HRESULT indicating the result of previous operations (If SUCCEEDED(hrPrev) equals false, no operation is executed.) *)
	END_VAR

END_FUNCTION

// Functions/Basic Image Operations/F_VN_CopyImageRegion

	{attribute 'TcIecLibraryType'}
	{attribute 'external_name' := 'F_VN_CopyImageRegion_GUID_9361A561_4665_D41E_957A_9C22A84B6A3B'}
	(* Deep copy the specified region of interest into a new image. *)
	FUNCTION F_VN_CopyImageRegion : HRESULT
	VAR_INPUT
		ipSrcImage	:	ITcVnImage;	(* Source image *)
		nX	:	UDINT;	(* Left boundary (inclusive 0-based index) *)
		nY	:	UDINT;	(* Upper boundary (inclusive 0-based index) *)
		nWidth	:	UDINT;	(* ROI width *)
		nHeight	:	UDINT;	(* ROI height *)
		ipDestImage	:	REFERENCE TO ITcVnImage;	(* Destination image (An appropriate destination image will be created if required.) *)
		hrPrev	:	HRESULT;	(* HRESULT indicating the result of previous operations (If SUCCEEDED(hrPrev) equals false, no operation is executed.) *)
	END_VAR

END_FUNCTION

// Functions/Basic Image Operations/F_VN_CopyImageRegionToRegion

	{attribute 'TcIecLibraryType'}
	{attribute 'external_name' := 'F_VN_CopyImageRegionToRegion_GUID_044EA8E5_1ACE_D6AF_BF59_8F9457710A41'}
	(* Copy an image region into another image region. *)
	FUNCTION F_VN_CopyImageRegionToRegion : HRESULT
	VAR_INPUT
		ipSrcImage	:	ITcVnImage;	(* Source image *)
		nXSrc	:	UDINT;	(* Left boundary in ipSrcImage (inclusive 0-based index) *)
		nYSrc	:	UDINT;	(* Upper boundary in ipSrcImage (inclusive 0-based index) *)
		nWidth	:	UDINT;	(* ROI width *)
		nHeight	:	UDINT;	(* ROI height *)
		ipDestImage	:	ITcVnImage;	(* Destination image (same type as ipSrcImage) *)
		nXDest	:	UDINT;	(* Left boundary in ipDestImage (inclusive 0-based index) *)
		nYDest	:	UDINT;	(* Upper boundary in ipDestImage (inclusive 0-based index) *)
		hrPrev	:	HRESULT;	(* HRESULT indicating the result of previous operations (If SUCCEEDED(hrPrev) equals false, no operation is executed.) *)
	END_VAR

END_FUNCTION

// Functions/Basic Image Operations/F_VN_CopyIntoDisplayableImage

	{attribute 'TcIecLibraryType'}
	{attribute 'external_name' := 'F_VN_CopyIntoDisplayableImage_GUID_00DB8C16_2B7D_D59C_A39C_37075511132D'}
	(* Copys an image into a displayable image. If you do not want to use ipSrcImage after this function call, you might want to use F_VN_TransformIntoDisplayableImage instead for better performance. *)
	FUNCTION F_VN_CopyIntoDisplayableImage : HRESULT
	VAR_INPUT
		ipSrcImage	:	ITcVnImage;	(* Source image *)
		ipDestImage	:	REFERENCE TO ITcVnDisplayableImage;	(* Returns the displayable image *)
		hrPrev	:	HRESULT;	(* HRESULT indicating the result of previous operations (If SUCCEEDED(hrPrev) equals false, no operation is executed.) *)
	END_VAR

END_FUNCTION

// Functions/Basic Image Operations/F_VN_TransformIntoDisplayableImage

	{attribute 'TcIecLibraryType'}
	{attribute 'external_name' := 'F_VN_TransformIntoDisplayableImage_GUID_F1551419_7157_D6BC_B4F2_4879CE3D1598'}
	(* Transform an image into a displayable image. The source image will be released and zeroed while existing destination images will be released and overwritten with the function result. The source image must not be used anywhere else and the transformation is very fast. If you want to use ipSrcImage after this function call, use F_VN_CopyIntoDisplayableImage instead. *)
	FUNCTION F_VN_TransformIntoDisplayableImage : HRESULT
	VAR_INPUT
		ipSrcImage	:	REFERENCE TO ITcVnImage;	(* Source image *)
		ipDestImage	:	REFERENCE TO ITcVnDisplayableImage;	(* Returns the displayable image *)
		hrPrev	:	HRESULT;	(* HRESULT indicating the result of previous operations (If SUCCEEDED(hrPrev) equals false, no operation is executed.) *)
	END_VAR

END_FUNCTION

// Functions/Basic Image Operations/F_VN_CreateAssociatedImage

	{attribute 'TcIecLibraryType'}
	{attribute 'external_name' := 'F_VN_CreateAssociatedImage_GUID_B36646F1_9137_D7FE_81BB_2CA4340FD8B3'}
	(* Creates a new image that shares its data with the source image. E.g. useful to work on different (disjoint) ROIs in parallel. *)
	FUNCTION F_VN_CreateAssociatedImage : HRESULT
	VAR_INPUT
		ipSrcImage	:	ITcVnImage;	(* Source image *)
		ipDestImage	:	REFERENCE TO ITcVnImage;	(* Returns the created image (Non-zero interface pointers are reused.) *)
		hrPrev	:	HRESULT;	(* HRESULT indicating the result of previous operations (If SUCCEEDED(hrPrev) equals false, no operation is executed.) *)
	END_VAR

END_FUNCTION

// Functions/Basic Image Operations/F_VN_CreateEmptyImage

	{attribute 'TcIecLibraryType'}
	{attribute 'external_name' := 'F_VN_CreateEmptyImage_GUID_746BD346_10BE_D78F_BE9C_CBC2604BB7C0'}
	(* Creates an empty image without allocating any data buffer. The initial reference count is set to one if a new image interface is created and kept, otherwise. *)
	FUNCTION F_VN_CreateEmptyImage : HRESULT
	VAR_INPUT
		ipImage	:	REFERENCE TO ITcVnImage;	(* Returns the created image *)
		hrPrev	:	HRESULT;	(* HRESULT indicating the result of previous operations (If SUCCEEDED(hrPrev) equals false, no operation is executed.) *)
	END_VAR

END_FUNCTION

// Functions/Basic Image Operations/F_VN_CreateImage

	{attribute 'TcIecLibraryType'}
	{attribute 'external_name' := 'F_VN_CreateImage_GUID_7EC1D48C_D2EE_DF6F_88E3_43DE8333BFBB'}
	(* Creates an image and allocate an appropriate data buffer. The initial reference count is set to one if a new image interface is created and kept, otherwise. *)
	FUNCTION F_VN_CreateImage : HRESULT
	VAR_INPUT
		ipImage	:	REFERENCE TO ITcVnImage;	(* Returns the created image (Non-zero interface pointers are reused.) *)
		nWidth	:	UDINT;	(* Image width *)
		nHeight	:	UDINT;	(* Image height *)
		ePixelType	:	ETcVnElementType;	(* Pixel type *)
		nChannelNum	:	UDINT;	(* Number of channels (1 to 255) *)
		hrPrev	:	HRESULT;	(* HRESULT indicating the result of previous operations (If SUCCEEDED(hrPrev) equals false, no operation is executed.) *)
	END_VAR

END_FUNCTION

// Functions/Basic Image Operations/F_VN_CreateNDimensionalImage

	{attribute 'TcIecLibraryType'}
	{attribute 'external_name' := 'F_VN_CreateNDimensionalImage_GUID_766FF9AB_383C_DC60_8501_0570F78A46E9'}
	(* Creates an N-dimensional image and allocates an appropriate data buffer. The initial reference count is set to one if a new image interface is created and kept, otherwise. *)
	FUNCTION F_VN_CreateNDimensionalImage : HRESULT
	VAR_INPUT
		ipImage	:	REFERENCE TO ITcVnImage;	(* Returns the created image (Non-zero interface pointers are reused.) *)
	END_VAR
	VAR_IN_OUT
		aShape	:	TcVnArray33_UDINT;	(* Specifies the shape of ipDestImage. First entry is the number of dimensions of ipImage (max. 32), followed by the sizes of each dimension. *)
	END_VAR
	VAR_INPUT
		ePixelType	:	ETcVnElementType;	(* Pixel type *)
		hrPrev	:	HRESULT;	(* HRESULT indicating the result of previous operations (If SUCCEEDED(hrPrev) equals false, no operation is executed.) *)
	END_VAR

END_FUNCTION

// Functions/Basic Image Operations/F_VN_CreateImageAndSetPixels

	{attribute 'TcIecLibraryType'}
	{attribute 'external_name' := 'F_VN_CreateImageAndSetPixels_GUID_5B27FBA9_3248_D660_8971_03B6F78E3A72'}
	(* Creates an image, allocates an appropriate data buffer and sets all pixels to the specified value. The initial reference count is set to one if a new image interface is created and kept, otherwise. *)
	FUNCTION F_VN_CreateImageAndSetPixels : HRESULT
	VAR_INPUT
		ipImage	:	REFERENCE TO ITcVnImage;	(* Returns the created image (Non-zero interface pointers are reused.) *)
		nWidth	:	UDINT;	(* Image width *)
		nHeight	:	UDINT;	(* Image height *)
		ePixelType	:	ETcVnElementType;	(* Pixel type *)
		nChannelNum	:	UDINT;	(* Number of channels (1 to 4) *)
	END_VAR
	VAR_IN_OUT
		aValue	:	TcVnVector4_LREAL;	(* Pixel value *)
	END_VAR
	VAR_INPUT
		hrPrev	:	HRESULT;	(* HRESULT indicating the result of previous operations (If SUCCEEDED(hrPrev) equals false, no operation is executed.) *)
	END_VAR

END_FUNCTION

// Functions/Basic Image Operations/F_VN_CreateNDimensionalImageAndSetPixels

	{attribute 'TcIecLibraryType'}
	{attribute 'external_name' := 'F_VN_CreateNDimensionalImageAndSetPixels_GUID_4C564B05_4BF8_D5C9_90CA_BAFD14CD89A0'}
	(* Creates an N-dimensional image, allocates an appropriate data buffer and sets all pixels to the specified value. The initial reference count is set to one if a new image interface is created and kept, otherwise. *)
	FUNCTION F_VN_CreateNDimensionalImageAndSetPixels : HRESULT
	VAR_INPUT
		ipImage	:	REFERENCE TO ITcVnImage;	(* Returns the created image (Non-zero interface pointers are reused.) *)
	END_VAR
	VAR_IN_OUT
		aShape	:	TcVnArray33_UDINT;	(* Specifies the shape of ipDestImage. First entry is the number of dimensions of ipImage (max. 32), followed by the sizes of each dimension. *)
	END_VAR
	VAR_INPUT
		ePixelType	:	ETcVnElementType;	(* Pixel type *)
		fValue	:	LREAL;	(* Pixel value *)
		hrPrev	:	HRESULT;	(* HRESULT indicating the result of previous operations (If SUCCEEDED(hrPrev) equals false, no operation is executed.) *)
	END_VAR

END_FUNCTION

// Functions/Basic Image Operations/F_VN_CreateImageFromArray

	{attribute 'TcIecLibraryType'}
	{attribute 'external_name' := 'F_VN_CreateImageFromArray_GUID_9278296F_ACD8_DA0A_88D4_8FA44DD493DD'}
	(* Creates an image and initialize it with the provided data. The initial reference count is set to one if a new image interface is created and kept, otherwise. *)
	FUNCTION F_VN_CreateImageFromArray : HRESULT
	VAR_INPUT
		pData	:	PVOID;	(* Pointer to the 1D data array. Make sure that the array contains at least nWidth * nHeight * nChannelNum elements and that the array element type matches ePixelType. *)
		ipImage	:	REFERENCE TO ITcVnImage;	(* Returns the created image (Non-zero interface pointers are reused.) *)
		nWidth	:	UDINT;	(* Image width *)
		nHeight	:	UDINT;	(* Image height *)
		ePixelType	:	ETcVnElementType;	(* Pixel type *)
		nChannelNum	:	UDINT;	(* Number of channels (1 to 255) *)
		hrPrev	:	HRESULT;	(* HRESULT indicating the result of previous operations (If SUCCEEDED(hrPrev) equals false, no operation is executed.) *)
	END_VAR

END_FUNCTION

// Functions/Basic Image Operations/F_VN_CreateNDimensionalImageFromArray

	{attribute 'TcIecLibraryType'}
	{attribute 'external_name' := 'F_VN_CreateNDimensionalImageFromArray_GUID_6C785C16_C171_D1D2_845A_5FD7A51CD4E3'}
	(* Creates an N-dimensional image and initialize it with the provided data. The initial reference count is set to one if a new image interface is created and kept, otherwise. *)
	FUNCTION F_VN_CreateNDimensionalImageFromArray : HRESULT
	VAR_INPUT
		pData	:	PVOID;	(* Pointer to the 1D data array. Ensure that the array contains at least the number of elements equal to the product of all dimensions in aShape and that the array element type matches ePixelType. *)
		ipImage	:	REFERENCE TO ITcVnImage;	(* Returns the created image (Non-zero interface pointers are reused.) *)
	END_VAR
	VAR_IN_OUT
		aShape	:	TcVnArray33_UDINT;	(* Specifies the shape of ipDestImage. First entry is the number of dimensions of ipImage (max. 32), followed by the sizes of each dimension. *)
	END_VAR
	VAR_INPUT
		ePixelType	:	ETcVnElementType;	(* Pixel type *)
		hrPrev	:	HRESULT;	(* HRESULT indicating the result of previous operations (If SUCCEEDED(hrPrev) equals false, no operation is executed.) *)
	END_VAR

END_FUNCTION

// Functions/Basic Image Operations/F_VN_ExportImage

	{attribute 'TcIecLibraryType'}
	{attribute 'external_name' := 'F_VN_ExportImage_GUID_E1268AFA_B932_D368_835B_C464F7CF0C8E'}
	(* Exports the image data into a given buffer (e.g. an array). F_VN_ExportImageSize should be called before to get the required buffer size. *)
	FUNCTION F_VN_ExportImage : HRESULT
	VAR_INPUT
		ipImage	:	ITcVnImage;	(* Image *)
		pBuffer	:	PVOID;	(* Pointer to a buffer to store the image data (Make sure to allocate enough memory! The required size in bytes can be determined using the function F_VN_ExportImageSize) *)
		nBufferSize	:	ULINT;	(* Size of the buffer memory in bytes *)
		hrPrev	:	HRESULT;	(* HRESULT indicating the result of previous operations (If SUCCEEDED(hrPrev) equals false, no operation is executed.) *)
	END_VAR

END_FUNCTION

// Functions/Basic Image Operations/F_VN_ExportImageSize

	{attribute 'TcIecLibraryType'}
	{attribute 'external_name' := 'F_VN_ExportImageSize_GUID_6A99F40C_4BE5_DC2B_A439_020A9CF353CD'}
	(* Get the required buffer size (in bytes) to store the image data. *)
	FUNCTION F_VN_ExportImageSize : HRESULT
	VAR_INPUT
		ipImage	:	ITcVnImage;	(* Image *)
	END_VAR
	VAR_IN_OUT
		nBufferSize	:	ULINT;	(* Returns the required buffer size in bytes *)
	END_VAR
	VAR_INPUT
		hrPrev	:	HRESULT;	(* HRESULT indicating the result of previous operations (If SUCCEEDED(hrPrev) equals false, no operation is executed.) *)
	END_VAR

END_FUNCTION

// Functions/Basic Image Operations/F_VN_ExportImageAsBmp

	{attribute 'TcIecLibraryType'}
	{attribute 'external_name' := 'F_VN_ExportImageAsBmp_GUID_B87F7DD5_6DA6_DDD2_AD9C_7A89E3609FF6'}
	(* Exports the image as bitmap into a given buffer (e.g. an array). F_VN_ExportImageAsBmpSize should be called before to get the required buffer size. *)
	FUNCTION F_VN_ExportImageAsBmp : HRESULT
	VAR_INPUT
		ipImage	:	ITcVnImage;	(* Image *)
		pBuffer	:	PVOID;	(* Pointer to a buffer to store the bitmap image (Make sure to allocate enough memory! The required size in bytes can be determined using the function F_VN_ExportImageAsBmpSize) *)
		nBufferSize	:	ULINT;	(* Size of the buffer memory in bytes *)
		hrPrev	:	HRESULT;	(* HRESULT indicating the result of previous operations (If SUCCEEDED(hrPrev) equals false, no operation is executed.) *)
	END_VAR

END_FUNCTION

// Functions/Basic Image Operations/F_VN_ExportImageAsBmpSize

	{attribute 'TcIecLibraryType'}
	{attribute 'external_name' := 'F_VN_ExportImageAsBmpSize_GUID_FC6C04EC_634C_D0BF_B7A5_C19FA207A2BA'}
	(* Get the required buffer size (in bytes) to store the image as bitmap. *)
	FUNCTION F_VN_ExportImageAsBmpSize : HRESULT
	VAR_INPUT
		ipImage	:	ITcVnImage;	(* Image *)
	END_VAR
	VAR_IN_OUT
		nBufferSize	:	ULINT;	(* Returns the required buffer size in bytes *)
	END_VAR
	VAR_INPUT
		hrPrev	:	HRESULT;	(* HRESULT indicating the result of previous operations (If SUCCEEDED(hrPrev) equals false, no operation is executed.) *)
	END_VAR

END_FUNCTION

// Functions/Basic Image Operations/F_VN_ExportImageAsBmpExp

	{attribute 'TcIecLibraryType'}
	{attribute 'external_name' := 'F_VN_ExportImageAsBmpExp_GUID_B4C6E9E7_6E92_D48F_9E46_193216933860'}
	(* Exports the image as bitmap into a given buffer (e.g. an array). F_VN_ExportImageAsBmpSizeExp should be called before to get the required buffer size. (expert function) *)
	FUNCTION F_VN_ExportImageAsBmpExp : HRESULT
	VAR_INPUT
		ipImage	:	ITcVnImage;	(* Image *)
		pBuffer	:	PVOID;	(* Pointer to a buffer to store the bitmap image (Make sure to allocate enough memory! The required size in bytes can be determined using the function F_VN_ExportImageAsBmpSizeExp) *)
		nBufferSize	:	ULINT;	(* Size of the buffer memory in bytes *)
		nWidth	:	UDINT;	(* Desired width (or 0 to keep the original width) *)
		nHeight	:	UDINT;	(* Desired height (or 0 to keep the original height) *)
		hrPrev	:	HRESULT;	(* HRESULT indicating the result of previous operations (If SUCCEEDED(hrPrev) equals false, no operation is executed.) *)
	END_VAR

END_FUNCTION

// Functions/Basic Image Operations/F_VN_ExportImageAsBmpSizeExp

	{attribute 'TcIecLibraryType'}
	{attribute 'external_name' := 'F_VN_ExportImageAsBmpSizeExp_GUID_E69F7422_AD5B_D61A_A25C_1A5257E0009E'}
	(* Get the required buffer size (in bytes) to store the image as bitmap. (expert function) *)
	FUNCTION F_VN_ExportImageAsBmpSizeExp : HRESULT
	VAR_INPUT
		ipImage	:	ITcVnImage;	(* Image *)
	END_VAR
	VAR_IN_OUT
		nBufferSize	:	ULINT;	(* Returns the required buffer size in bytes *)
	END_VAR
	VAR_INPUT
		nWidth	:	UDINT;	(* Desired width (or 0 to keep the original width) *)
		nHeight	:	UDINT;	(* Desired height (or 0 to keep the original height) *)
		hrPrev	:	HRESULT;	(* HRESULT indicating the result of previous operations (If SUCCEEDED(hrPrev) equals false, no operation is executed.) *)
	END_VAR

END_FUNCTION

// Functions/Basic Image Operations/F_VN_FuseImages

	{attribute 'TcIecLibraryType'}
	{attribute 'external_name' := 'F_VN_FuseImages_GUID_B742C2C2_206D_D337_BCD9_55BA445341FC'}
	(* Fuse 2 images vertically (intended for line scan cameras). *)
	FUNCTION F_VN_FuseImages : HRESULT
	VAR_INPUT
		ipSrcImage1	:	ITcVnImage;	(* Source image 1 *)
		ipSrcImage2	:	ITcVnImage;	(* Source image 2 *)
		ipDestImage	:	REFERENCE TO ITcVnImage;	(* Destination image *)
		nFirstLine	:	UDINT;	(* Line index in ipSrcImage1, which is the first line in ipDestImage *)
		nNumLines	:	UDINT;	(* The number of lines that should be copied to ipDestImage, starting with nFirstLine in ipSrcImage1. Once the last line of ipSrcImage1 was copied, the remaining lines are copied from ipSrcImage2, starting at line index 0. *)
		hrPrev	:	HRESULT;	(* HRESULT indicating the result of previous operations (If SUCCEEDED(hrPrev) equals false, no operation is executed.) *)
	END_VAR

END_FUNCTION

// Functions/Basic Image Operations/F_VN_FuseImagesArray

	{attribute 'TcIecLibraryType'}
	{attribute 'external_name' := 'F_VN_FuseImagesArray_GUID_834BA529_38FC_D43A_B832_5A8E7D3294B6'}
	(* Fuse up to 10 images vertically (intended for line scan cameras). *)
	FUNCTION F_VN_FuseImagesArray : HRESULT
	VAR_IN_OUT
		aSrcImageArray	:	TcVnArray10_ITcVnImage;	(* Ten-element source image array (not all elements need to be filled, nValidImages specifies the actual amount of images) *)
	END_VAR
	VAR_INPUT
		nValidImages	:	UDINT;	(* Number of valid images in aSrcImageArray *)
		ipDestImage	:	REFERENCE TO ITcVnImage;	(* Destination image *)
		nFirstLine	:	UDINT;	(* Line index in ipSrcImage1, which is the first line in ipDestImage *)
		nNumLines	:	UDINT;	(* The number of lines that should be copied to ipDestImage, starting with nFirstLine in aSrcImageArray[0]. Once the last line of aSrcImageArray[0] was copied, the remaining lines are copied from aSrcImageArray[1] (starting at line index 0) and so on. *)
		hrPrev	:	HRESULT;	(* HRESULT indicating the result of previous operations (If SUCCEEDED(hrPrev) equals false, no operation is executed.) *)
	END_VAR

END_FUNCTION

// Functions/Basic Image Operations/F_VN_GetImageChannel

	{attribute 'TcIecLibraryType'}
	{attribute 'external_name' := 'F_VN_GetImageChannel_GUID_E6ACD7D5_00F7_D0BC_85A5_E098DDDA2C45'}
	(* Return the specified source image channel as a single-channel image. *)
	FUNCTION F_VN_GetImageChannel : HRESULT
	VAR_INPUT
		ipSrcImage	:	ITcVnImage;	(* Source image *)
		ipDestImage	:	REFERENCE TO ITcVnImage;	(* Destination image (An appropriate image will be created if required.) *)
		nChannelIndex	:	UINT;	(* Index of the requested source image channel *)
		hrPrev	:	HRESULT;	(* HRESULT indicating the result of previous operations (If SUCCEEDED(hrPrev) equals false, no operation is executed.) *)
	END_VAR

END_FUNCTION

// Functions/Basic Image Operations/F_VN_GetImageHeight

	{attribute 'TcIecLibraryType'}
	{attribute 'external_name' := 'F_VN_GetImageHeight_GUID_966A1794_07DD_D3D4_8BE6_20B45108551D'}
	(* Return the height of an image. (Alternatively use interface method .GetHeight.) *)
	FUNCTION F_VN_GetImageHeight : HRESULT
	VAR_INPUT
		ipImage	:	ITcVnImage;	(* Image *)
	END_VAR
	VAR_IN_OUT
		nHeight	:	UDINT;	(* Return the height of ipImage *)
	END_VAR
	VAR_INPUT
		hrPrev	:	HRESULT;	(* HRESULT indicating the result of previous operations (If SUCCEEDED(hrPrev) equals false, no operation is executed.) *)
	END_VAR

END_FUNCTION

// Functions/Basic Image Operations/F_VN_GetImageInfo

	{attribute 'TcIecLibraryType'}
	{attribute 'external_name' := 'F_VN_GetImageInfo_GUID_D7279982_43B9_D458_9A08_1AFDE776886E'}
	(* Gets a struct containing all common meta infos of the image. (Alternatively use interface method .GetImageInfo.) *)
	FUNCTION F_VN_GetImageInfo : HRESULT
	VAR_INPUT
		ipImage	:	ITcVnImage;	(* Image *)
	END_VAR
	VAR_IN_OUT
		stImageInfo	:	TcVnImageInfo;	(* Returns a struct describing the image *)
	END_VAR
	VAR_INPUT
		hrPrev	:	HRESULT;	(* HRESULT indicating the result of previous operations (If SUCCEEDED(hrPrev) equals false, no operation is executed.) *)
	END_VAR

END_FUNCTION

// Functions/Basic Image Operations/F_VN_GetImageWidth

	{attribute 'TcIecLibraryType'}
	{attribute 'external_name' := 'F_VN_GetImageWidth_GUID_AE88EBF3_32EF_DFD2_9732_BBDBD198CEF7'}
	(* Return the width of an image. (Alternatively use interface method .GetWidth.) *)
	FUNCTION F_VN_GetImageWidth : HRESULT
	VAR_INPUT
		ipImage	:	ITcVnImage;	(* Image *)
	END_VAR
	VAR_IN_OUT
		nWidth	:	UDINT;	(* Return the width of ipImage *)
	END_VAR
	VAR_INPUT
		hrPrev	:	HRESULT;	(* HRESULT indicating the result of previous operations (If SUCCEEDED(hrPrev) equals false, no operation is executed.) *)
	END_VAR

END_FUNCTION

// Functions/Basic Image Operations/F_VN_GetLayoutInfo

	{attribute 'TcIecLibraryType'}
	{attribute 'external_name' := 'F_VN_GetLayoutInfo_GUID_21E34241_84E1_D06C_AF3A_D66F6F2FD631'}
	(* Return the layout information of an image *)
	FUNCTION F_VN_GetLayoutInfo : HRESULT
	VAR_INPUT
		ipImage	:	ITcVnImage;	(* Source image *)
	END_VAR
	VAR_IN_OUT
		aLayoutInfo	:	TcVnArray33_UDINT;	(* Contains layout information of ipImage. First entry of the aLayoutInfo is the number of dimensions of ipImage (max. 32), followed by the sizes of each dimension. *)
	END_VAR
	VAR_INPUT
		hrPrev	:	HRESULT;	(* HRESULT indicating the result of previous operations (If SUCCEEDED(hrPrev) equals false, no operation is executed.) *)
	END_VAR

END_FUNCTION

// Functions/Basic Image Operations/F_VN_GetPixel

	{attribute 'TcIecLibraryType'}
	{attribute 'external_name' := 'F_VN_GetPixel_GUID_AC61E7CB_3CBE_D5B2_806B_0036F690DED2'}
	(* Gets a specific pixel. *)
	FUNCTION F_VN_GetPixel : HRESULT
	VAR_INPUT
		ipSrcImage	:	ITcVnImage;	(* Source image *)
	END_VAR
	VAR_IN_OUT
		aValue	:	TcVnVector4_LREAL;	(* Returns the pixel value (Unused channels are set to 0.) *)
	END_VAR
	VAR_INPUT
		nX	:	UDINT;	(* x coordinate of the pixel *)
		nY	:	UDINT;	(* y coordinate of the pixel *)
		hrPrev	:	HRESULT;	(* HRESULT indicating the result of previous operations (If SUCCEEDED(hrPrev) equals false, no operation is executed.) *)
	END_VAR

END_FUNCTION

// Functions/Basic Image Operations/F_VN_GetPixelFormat

	{attribute 'TcIecLibraryType'}
	{attribute 'external_name' := 'F_VN_GetPixelFormat_GUID_2769E23D_10CB_D25A_B863_EA3F2BDDF851'}
	(* Gets the pixel format of an image. (Alternatively use interface method .GetPixelFormat.) *)
	FUNCTION F_VN_GetPixelFormat : HRESULT
	VAR_INPUT
		ipImage	:	ITcVnImage;	(* Image *)
	END_VAR
	VAR_IN_OUT
		stPixelFormat	:	TcVnPixelFormat;	(* Returns a struct describing the pixel format *)
	END_VAR
	VAR_INPUT
		hrPrev	:	HRESULT;	(* HRESULT indicating the result of previous operations (If SUCCEEDED(hrPrev) equals false, no operation is executed.) *)
	END_VAR

END_FUNCTION

// Functions/Basic Image Operations/F_VN_GetRoi

	{attribute 'TcIecLibraryType'}
	{attribute 'external_name' := 'F_VN_GetRoi_GUID_E4CD7798_BA5E_D65D_8319_626E2FC7251B'}
	(* Gets the coordinates of the region of interest (ROI) within the image. *)
	FUNCTION F_VN_GetRoi : HRESULT
	VAR_INPUT
		ipSrcImage	:	ITcVnImage;	(* Source image *)
	END_VAR
	VAR_IN_OUT
		stRoi	:	TcVnRectangle_UDINT;	(* Returns the coordinates of the region of interest *)
	END_VAR
	VAR_INPUT
		hrPrev	:	HRESULT;	(* HRESULT indicating the result of previous operations (If SUCCEEDED(hrPrev) equals false, no operation is executed.) *)
	END_VAR

END_FUNCTION

// Functions/Basic Image Operations/F_VN_MixImageChannels

	{attribute 'TcIecLibraryType'}
	{attribute 'external_name' := 'F_VN_MixImageChannels_GUID_E24DD01C_85A3_DC4D_A106_EFBD0E093729'}
	(* Mix image channels by copying the specified channels of the source image into the specified channels of the destination image. *)
	FUNCTION F_VN_MixImageChannels : HRESULT
	VAR_INPUT
		ipSrcImage	:	ITcVnImage;	(* Source image *)
		ipDestImage	:	REFERENCE TO ITcVnImage;	(* Destination image (An appropriate image will be created if required.) *)
		ipIndicesFromTo	:	ITcVnContainer;	(* Index pairs (ContainerType_Vector_TcVnVector2_DINT), specifying which source channel (TcVnVector2_DINT [0]) should be copied to which destination channel (TcVnVector2_DINT [1]). *)
		hrPrev	:	HRESULT;	(* HRESULT indicating the result of previous operations (If SUCCEEDED(hrPrev) equals false, no operation is executed.) *)
	END_VAR

END_FUNCTION

// Functions/Basic Image Operations/F_VN_PadImageBorder

	{attribute 'TcIecLibraryType'}
	{attribute 'external_name' := 'F_VN_PadImageBorder_GUID_1AC2DBAA_85AD_D005_8A00_3882B6E10806'}
	(* Add padding (zeros) around the original image borders. *)
	FUNCTION F_VN_PadImageBorder : HRESULT
	VAR_INPUT
		ipSrcImage	:	ITcVnImage;	(* Source image *)
		ipPaddedImage	:	REFERENCE TO ITcVnImage;	(* Padded destination image (Same type as ipSrcImage, an appropriate destination image will be created if required.) *)
		nTopBorder	:	UDINT;	(* Padding height in pixels above top border *)
		nBottomBorder	:	UDINT;	(* Padding height in pixels below bottom border *)
		nLeftBorder	:	UDINT;	(* Padding width in pixels before left border *)
		nRightBorder	:	UDINT;	(* Padding width in pixels after right border *)
		hrPrev	:	HRESULT;	(* HRESULT indicating the result of previous operations (If SUCCEEDED(hrPrev) equals false, no operation is executed.) *)
	END_VAR

END_FUNCTION

// Functions/Basic Image Operations/F_VN_PadImageBorderExp

	{attribute 'TcIecLibraryType'}
	{attribute 'external_name' := 'F_VN_PadImageBorderExp_GUID_BDE86C1D_B318_D522_88C2_CB950E237AAB'}
	(* Add padding around the original image borders. (expert function) *)
	FUNCTION F_VN_PadImageBorderExp : HRESULT
	VAR_INPUT
		ipSrcImage	:	ITcVnImage;	(* Source image *)
		ipPaddedImage	:	REFERENCE TO ITcVnImage;	(* Padded destination image (Same type as ipSrcImage, an appropriate destination image will be created if required.) *)
		nTopBorder	:	UDINT;	(* Padding height in pixels above top border *)
		nBottomBorder	:	UDINT;	(* Padding height in pixels below bottom border *)
		nLeftBorder	:	UDINT;	(* Padding width in pixels before left border *)
		nRightBorder	:	UDINT;	(* Padding width in pixels after right border *)
		ePaddingType	:	ETcVnBorderInterpolationMethod;	(* Specifies how the pixel values of the padding area are determined *)
	END_VAR
	VAR_IN_OUT
		aPaddingValue	:	TcVnVector4_LREAL;	(* Specifies the padding value if CONSTANT is used *)
	END_VAR
	VAR_INPUT
		hrPrev	:	HRESULT;	(* HRESULT indicating the result of previous operations (If SUCCEEDED(hrPrev) equals false, no operation is executed.) *)
	END_VAR

END_FUNCTION

// Functions/Basic Image Operations/F_VN_ReinterpretUnsupportedImage

	{attribute 'TcIecLibraryType'}
	{attribute 'external_name' := 'F_VN_ReinterpretUnsupportedImage_GUID_84DB0B90_553B_D197_8FE6_B5EEE9EC33C1'}
	(* Reinterpret an unsupported image using additional information. If successful, the image will be of a supported type. *)
	FUNCTION F_VN_ReinterpretUnsupportedImage : HRESULT
	VAR_INPUT
		ipImage	:	ITcVnImage;	(* Image to be reinterpreted *)
		ePixelType	:	ETcVnElementType;	(* Pixel element type to be used for reinterpreting the image data *)
		hrPrev	:	HRESULT;	(* HRESULT indicating the result of previous operations (If SUCCEEDED(hrPrev) equals false, no operation is executed.) *)
	END_VAR

END_FUNCTION

// Functions/Basic Image Operations/F_VN_ResetRoi

	{attribute 'TcIecLibraryType'}
	{attribute 'external_name' := 'F_VN_ResetRoi_GUID_345D44EF_9D88_D88E_9EE9_2E66A6EEC818'}
	(* Reset the region of interest (ROI) of an image. (After this operation, the ROI is set to the entire image.) *)
	FUNCTION F_VN_ResetRoi : HRESULT
	VAR_INPUT
		ipImage	:	ITcVnImage;	(* Image *)
		hrPrev	:	HRESULT;	(* HRESULT indicating the result of previous operations (If SUCCEEDED(hrPrev) equals false, no operation is executed.) *)
	END_VAR

END_FUNCTION

// Functions/Basic Image Operations/F_VN_SetImageChannel

	{attribute 'TcIecLibraryType'}
	{attribute 'external_name' := 'F_VN_SetImageChannel_GUID_121C6D16_C003_D1AE_B698_172F0A97081D'}
	(* Sets the specified destination image channel to the values of the specified source image channel. *)
	FUNCTION F_VN_SetImageChannel : HRESULT
	VAR_INPUT
		ipSrcImage	:	ITcVnImage;	(* Source image *)
		ipDestImage	:	REFERENCE TO ITcVnImage;	(* Destination image (An appropriate image will be created if required.) *)
		nSrcChannelIndex	:	UINT;	(* Index of the source image channel *)
		nDestChannelIndex	:	UINT;	(* Index of the destination image channel, which will be replaced by the specified source image channel *)
		hrPrev	:	HRESULT;	(* HRESULT indicating the result of previous operations (If SUCCEEDED(hrPrev) equals false, no operation is executed.) *)
	END_VAR

END_FUNCTION

// Functions/Basic Image Operations/F_VN_SetPixel

	{attribute 'TcIecLibraryType'}
	{attribute 'external_name' := 'F_VN_SetPixel_GUID_9349450F_9A4F_D5F4_919E_BC6E52DC112E'}
	(* Sets a specific pixel. *)
	FUNCTION F_VN_SetPixel : HRESULT
	VAR_INPUT
		ipSrcImage	:	ITcVnImage;	(* Source image *)
	END_VAR
	VAR_IN_OUT
		aValue	:	TcVnVector4_LREAL;	(* The pixel value to set (additional channels are ignored.) *)
	END_VAR
	VAR_INPUT
		nX	:	UDINT;	(* x coordinate of the pixel *)
		nY	:	UDINT;	(* y coordinate of the pixel *)
		hrPrev	:	HRESULT;	(* HRESULT indicating the result of previous operations (If SUCCEEDED(hrPrev) equals false, no operation is executed.) *)
	END_VAR

END_FUNCTION

// Functions/Basic Image Operations/F_VN_SetPixels

	{attribute 'TcIecLibraryType'}
	{attribute 'external_name' := 'F_VN_SetPixels_GUID_E2EE67EB_FE9E_DB30_9775_A63073DF3A11'}
	(* Sets all pixels of an image to a given value. *)
	FUNCTION F_VN_SetPixels : HRESULT
	VAR_INPUT
		ipDestImage	:	ITcVnImage;	(* Destination image *)
	END_VAR
	VAR_IN_OUT
		aValue	:	TcVnVector4_LREAL;	(* Pixel value *)
	END_VAR
	VAR_INPUT
		hrPrev	:	HRESULT;	(* HRESULT indicating the result of previous operations (If SUCCEEDED(hrPrev) equals false, no operation is executed.) *)
	END_VAR

END_FUNCTION

// Functions/Basic Image Operations/F_VN_SetPixelsExp

	{attribute 'TcIecLibraryType'}
	{attribute 'external_name' := 'F_VN_SetPixelsExp_GUID_5DC679A4_D8B3_D79C_83EC_5328B55D9F8B'}
	(* Sets all pixels of an image to a given value. (expert function) *)
	FUNCTION F_VN_SetPixelsExp : HRESULT
	VAR_INPUT
		ipDestImage	:	ITcVnImage;	(* Destination image *)
	END_VAR
	VAR_IN_OUT
		aValue	:	TcVnVector4_LREAL;	(* Pixel value *)
	END_VAR
	VAR_INPUT
		ipMask	:	ITcVnImage;	(* Mask image *)
		hrPrev	:	HRESULT;	(* HRESULT indicating the result of previous operations (If SUCCEEDED(hrPrev) equals false, no operation is executed.) *)
	END_VAR

END_FUNCTION

// Functions/Basic Image Operations/F_VN_SetRoi

	{attribute 'TcIecLibraryType'}
	{attribute 'external_name' := 'F_VN_SetRoi_GUID_7352D3E1_4861_D1EF_8B71_95F582C5622B'}
	(* Sets a region of interest (ROI) within an image. *)
	FUNCTION F_VN_SetRoi : HRESULT
	VAR_INPUT
		nX	:	UDINT;	(* Left boundary (inclusive 0-based index) *)
		nY	:	UDINT;	(* Upper boundary (inclusive 0-based index) *)
		nWidth	:	UDINT;	(* ROI width *)
		nHeight	:	UDINT;	(* ROI height *)
		ipDestImage	:	ITcVnImage;	(* Destination image *)
		hrPrev	:	HRESULT;	(* HRESULT indicating the result of previous operations (If SUCCEEDED(hrPrev) equals false, no operation is executed.) *)
	END_VAR

END_FUNCTION

// Functions/Basic Image Operations/F_VN_SetRoi_TcVnRectangle_DINT

	{attribute 'TcIecLibraryType'}
	{attribute 'external_name' := 'F_VN_SetRoi_TcVnRectangle_DINT_GUID_2D199ECB_16DD_D725_922F_6D1CBE3B1A88'}
	(* Sets a region of interest (ROI) within an image. *)
	FUNCTION F_VN_SetRoi_TcVnRectangle_DINT : HRESULT
	VAR_IN_OUT
		stRoi	:	TcVnRectangle_DINT;	(* Region of interest *)
	END_VAR
	VAR_INPUT
		ipDestImage	:	ITcVnImage;	(* Destination image *)
		hrPrev	:	HRESULT;	(* HRESULT indicating the result of previous operations (If SUCCEEDED(hrPrev) equals false, no operation is executed.) *)
	END_VAR

END_FUNCTION

// Functions/Basic Image Operations/F_VN_SetRoi_TcVnRectangle_UDINT

	{attribute 'TcIecLibraryType'}
	{attribute 'external_name' := 'F_VN_SetRoi_TcVnRectangle_UDINT_GUID_7823DD93_BD89_DD94_958C_BC5EF174191A'}
	(* Sets a region of interest (ROI) within an image. *)
	FUNCTION F_VN_SetRoi_TcVnRectangle_UDINT : HRESULT
	VAR_IN_OUT
		stRoi	:	TcVnRectangle_UDINT;	(* Region of interest *)
	END_VAR
	VAR_INPUT
		ipDestImage	:	ITcVnImage;	(* Destination image *)
		hrPrev	:	HRESULT;	(* HRESULT indicating the result of previous operations (If SUCCEEDED(hrPrev) equals false, no operation is executed.) *)
	END_VAR

END_FUNCTION

// Functions/Basic Image Operations/F_VN_SplitImageChannels

	{attribute 'TcIecLibraryType'}
	{attribute 'external_name' := 'F_VN_SplitImageChannels_GUID_B153E69A_6DF9_DE01_8719_329BC106E3E2'}
	(* Split a multi-channel image into multiple single channel images (1 for each source image channel). *)
	FUNCTION F_VN_SplitImageChannels : HRESULT
	VAR_INPUT
		ipSrcImage	:	ITcVnImage;	(* Source image with multiple channels *)
		pDestImages	:	PVOID;	(* Pointer to an array of ITcVnImage (appropriate destination images will be created if required) *)
		nArraySize	:	UINT;	(* Number of pDestImages array elements (array must be >= ipSourceImage channels) *)
		hrPrev	:	HRESULT;	(* HRESULT indicating the result of previous operations (If SUCCEEDED(hrPrev) equals false, no operation is executed.) *)
	END_VAR
	VAR_OUTPUT
		nImageChannels	:	UINT;	(* Actual source image channels *)
	END_VAR

END_FUNCTION

// Functions/Basic Image Operations/F_VN_TransformIntoDisplayableImageExp

	{attribute 'TcIecLibraryType'}
	{attribute 'external_name' := 'F_VN_TransformIntoDisplayableImageExp_GUID_0E7724B2_81D8_D568_8D2D_8371B5789F95'}
	(* Transform an image into a displayable image. The source image will be released and zeroed while existing destination images will be released and overwritten with the function result. If bAllowDeepCopy equals false, the source image must not be used anywhere else and the transformation is always very fast. Otherwise, if bAllowDeepCopy equals true, a deep copy of the source image might be created if required, which will result in a longer execution time. If you want to use ipSrcImage after this function call, use F_VN_CopyIntoDisplayableImage instead. (expert function) *)
	FUNCTION F_VN_TransformIntoDisplayableImageExp : HRESULT
	VAR_INPUT
		ipSrcImage	:	REFERENCE TO ITcVnImage;	(* Source image *)
		ipDestImage	:	REFERENCE TO ITcVnDisplayableImage;	(* Returns the displayable image *)
		bAllowDeepCopy	:	BOOL;	(* Allow deep image copies, if required *)
		hrPrev	:	HRESULT;	(* HRESULT indicating the result of previous operations (If SUCCEEDED(hrPrev) equals false, no operation is executed.) *)
	END_VAR

END_FUNCTION

// Functions/Container Statistics/F_VN_ContainerAverage

	{attribute 'TcIecLibraryType'}
	{attribute 'external_name' := 'F_VN_ContainerAverage_GUID_B2858614_050B_D563_A66A_D6FA3407EB08'}
	(* Calculate the average of elements in a container. *)
	FUNCTION F_VN_ContainerAverage : HRESULT
	VAR_INPUT
		ipSrcContainer	:	ITcVnContainer;	(* Source container (Arithmetic, point and vector element types are supported. For points and vectors, the euclidean norm is used.) *)
	END_VAR
	VAR_IN_OUT
		fAverage	:	LREAL;	(* Returns the calculated average value *)
	END_VAR
	VAR_INPUT
		hrPrev	:	HRESULT;	(* HRESULT indicating the result of previous operations (If SUCCEEDED(hrPrev) equals false, no operation is executed.) *)
	END_VAR

END_FUNCTION

// Functions/Container Statistics/F_VN_ContainerAverageElementwise2

	{attribute 'TcIecLibraryType'}
	{attribute 'external_name' := 'F_VN_ContainerAverageElementwise2_GUID_BD9B364B_D592_D794_AFD0_52CC3C7C434A'}
	(* Calculate the elementwise average of 2D elements in a container. *)
	FUNCTION F_VN_ContainerAverageElementwise2 : HRESULT
	VAR_INPUT
		ipSrcContainer	:	ITcVnContainer;	(* Source container with 2D points or vectors *)
	END_VAR
	VAR_IN_OUT
		aAverage	:	TcVnVector2_LREAL;	(* Returns the calculated average values *)
	END_VAR
	VAR_INPUT
		hrPrev	:	HRESULT;	(* HRESULT indicating the result of previous operations (If SUCCEEDED(hrPrev) equals false, no operation is executed.) *)
	END_VAR

END_FUNCTION

// Functions/Container Statistics/F_VN_ContainerAverageElementwise3

	{attribute 'TcIecLibraryType'}
	{attribute 'external_name' := 'F_VN_ContainerAverageElementwise3_GUID_58F3ED65_D8EB_DDC5_8AF9_0337A8E4C728'}
	(* Calculate the elementwise average of 3D elements in a container. *)
	FUNCTION F_VN_ContainerAverageElementwise3 : HRESULT
	VAR_INPUT
		ipSrcContainer	:	ITcVnContainer;	(* Source container with 3D points or vectors *)
	END_VAR
	VAR_IN_OUT
		aAverage	:	TcVnVector3_LREAL;	(* Returns the calculated average values *)
	END_VAR
	VAR_INPUT
		hrPrev	:	HRESULT;	(* HRESULT indicating the result of previous operations (If SUCCEEDED(hrPrev) equals false, no operation is executed.) *)
	END_VAR

END_FUNCTION

// Functions/Container Statistics/F_VN_ContainerAverageElementwise4

	{attribute 'TcIecLibraryType'}
	{attribute 'external_name' := 'F_VN_ContainerAverageElementwise4_GUID_C6A1425F_6A5A_D431_A364_AA961AD2B64A'}
	(* Calculate the elementwise average of 4D elements in a container. *)
	FUNCTION F_VN_ContainerAverageElementwise4 : HRESULT
	VAR_INPUT
		ipSrcContainer	:	ITcVnContainer;	(* Source container with 4D vectors *)
	END_VAR
	VAR_IN_OUT
		aAverage	:	TcVnVector4_LREAL;	(* Returns the calculated average values *)
	END_VAR
	VAR_INPUT
		hrPrev	:	HRESULT;	(* HRESULT indicating the result of previous operations (If SUCCEEDED(hrPrev) equals false, no operation is executed.) *)
	END_VAR

END_FUNCTION

// Functions/Container Statistics/F_VN_ContainerAverageVariance

	{attribute 'TcIecLibraryType'}
	{attribute 'external_name' := 'F_VN_ContainerAverageVariance_GUID_E060EA5E_9591_D91D_A89E_7748093095A8'}
	(* Calculate the average and variance of elements in a container. *)
	FUNCTION F_VN_ContainerAverageVariance : HRESULT
	VAR_INPUT
		ipSrcContainer	:	ITcVnContainer;	(* Source container (Arithmetic, point and vector element types are supported. For points and vectors, the euclidean norm is used.) *)
	END_VAR
	VAR_IN_OUT
		fAverage	:	LREAL;	(* Returns the calculated average value *)
		fVariance	:	LREAL;	(* Returns the calculated variance value *)
	END_VAR
	VAR_INPUT
		hrPrev	:	HRESULT;	(* HRESULT indicating the result of previous operations (If SUCCEEDED(hrPrev) equals false, no operation is executed.) *)
	END_VAR

END_FUNCTION

// Functions/Container Statistics/F_VN_ContainerAverageVarianceElementwise2

	{attribute 'TcIecLibraryType'}
	{attribute 'external_name' := 'F_VN_ContainerAverageVarianceElementwise2_GUID_85D56815_4E7F_D2E8_A5C2_0A19D6C39C71'}
	(* Calculate the elementwise average and variance of 2D elements in a container. *)
	FUNCTION F_VN_ContainerAverageVarianceElementwise2 : HRESULT
	VAR_INPUT
		ipSrcContainer	:	ITcVnContainer;	(* Source container with 2D points or vectors *)
	END_VAR
	VAR_IN_OUT
		aAverage	:	TcVnVector2_LREAL;	(* Returns the calculated average values *)
		aVariance	:	TcVnVector2_LREAL;	(* Returns the calculated variance values *)
	END_VAR
	VAR_INPUT
		hrPrev	:	HRESULT;	(* HRESULT indicating the result of previous operations (If SUCCEEDED(hrPrev) equals false, no operation is executed.) *)
	END_VAR

END_FUNCTION

// Functions/Container Statistics/F_VN_ContainerAverageVarianceElementwise3

	{attribute 'TcIecLibraryType'}
	{attribute 'external_name' := 'F_VN_ContainerAverageVarianceElementwise3_GUID_E28EE6BA_FE0B_DA05_B05E_C79F8613734D'}
	(* Calculate the elementwise average and variance of 3D elements in a container. *)
	FUNCTION F_VN_ContainerAverageVarianceElementwise3 : HRESULT
	VAR_INPUT
		ipSrcContainer	:	ITcVnContainer;	(* Source container with 3D points or vectors *)
	END_VAR
	VAR_IN_OUT
		aAverage	:	TcVnVector3_LREAL;	(* Returns the calculated average values *)
		aVariance	:	TcVnVector3_LREAL;	(* Returns the calculated variance values *)
	END_VAR
	VAR_INPUT
		hrPrev	:	HRESULT;	(* HRESULT indicating the result of previous operations (If SUCCEEDED(hrPrev) equals false, no operation is executed.) *)
	END_VAR

END_FUNCTION

// Functions/Container Statistics/F_VN_ContainerAverageVarianceElementwise4

	{attribute 'TcIecLibraryType'}
	{attribute 'external_name' := 'F_VN_ContainerAverageVarianceElementwise4_GUID_1B13A526_4C6E_D4DC_99E6_96EEB3B36D01'}
	(* Calculate the elementwise average and variance of 4D elements in a container. *)
	FUNCTION F_VN_ContainerAverageVarianceElementwise4 : HRESULT
	VAR_INPUT
		ipSrcContainer	:	ITcVnContainer;	(* Source container with 4D vectors *)
	END_VAR
	VAR_IN_OUT
		aAverage	:	TcVnVector4_LREAL;	(* Returns the calculated average values *)
		aVariance	:	TcVnVector4_LREAL;	(* Returns the calculated variance values *)
	END_VAR
	VAR_INPUT
		hrPrev	:	HRESULT;	(* HRESULT indicating the result of previous operations (If SUCCEEDED(hrPrev) equals false, no operation is executed.) *)
	END_VAR

END_FUNCTION

// Functions/Container Statistics/F_VN_MaxElement

	{attribute 'TcIecLibraryType'}
	{attribute 'external_name' := 'F_VN_MaxElement_GUID_8B5E0475_1791_DBFE_898A_ABEA65DA121F'}
	(* Gets the maximum element of a container. *)
	FUNCTION F_VN_MaxElement : HRESULT
	VAR_INPUT
		ipSrcContainer	:	ITcVnContainer;	(* Source container (Arithmetic, point and vector element types are supported. For points and vectors, the euclidean norm is used.) *)
		ipDestIterator	:	REFERENCE TO ITcVnBidirectionalIterator;	(* Returns an iterator to the requested element *)
	END_VAR
	VAR_IN_OUT
		nIndex	:	ULINT;	(* Returns the position of the requested element within the container *)
	END_VAR
	VAR_INPUT
		hrPrev	:	HRESULT;	(* HRESULT indicating the result of previous operations (If SUCCEEDED(hrPrev) equals false, no operation is executed.) *)
	END_VAR

END_FUNCTION

// Functions/Container Statistics/F_VN_MedianElement

	{attribute 'TcIecLibraryType'}
	{attribute 'external_name' := 'F_VN_MedianElement_GUID_6B4BBBF6_03D0_D5BB_92F7_0B7FDFF93116'}
	(* Gets the median element of a container. *)
	FUNCTION F_VN_MedianElement : HRESULT
	VAR_INPUT
		ipSrcContainer	:	ITcVnContainer;	(* Source container (Arithmetic, point and vector element types are supported. For points and vectors, the euclidean norm is used.) *)
		ipDestIterator	:	REFERENCE TO ITcVnBidirectionalIterator;	(* Returns an iterator to the requested element *)
	END_VAR
	VAR_IN_OUT
		nIndex	:	ULINT;	(* Returns the position of the requested element within the container *)
	END_VAR
	VAR_INPUT
		hrPrev	:	HRESULT;	(* HRESULT indicating the result of previous operations (If SUCCEEDED(hrPrev) equals false, no operation is executed.) *)
	END_VAR

END_FUNCTION

// Functions/Container Statistics/F_VN_MinElement

	{attribute 'TcIecLibraryType'}
	{attribute 'external_name' := 'F_VN_MinElement_GUID_8D6E5915_13BC_D9CE_ADB8_07EE2FC80431'}
	(* Gets the minimum element of a container. *)
	FUNCTION F_VN_MinElement : HRESULT
	VAR_INPUT
		ipSrcContainer	:	ITcVnContainer;	(* Source container (Arithmetic, point and vector element types are supported. For points and vectors, the euclidean norm is used.) *)
		ipDestIterator	:	REFERENCE TO ITcVnBidirectionalIterator;	(* Returns an iterator to the requested element *)
	END_VAR
	VAR_IN_OUT
		nIndex	:	ULINT;	(* Returns the position of the requested element within the container *)
	END_VAR
	VAR_INPUT
		hrPrev	:	HRESULT;	(* HRESULT indicating the result of previous operations (If SUCCEEDED(hrPrev) equals false, no operation is executed.) *)
	END_VAR

END_FUNCTION

// Functions/Fourier Analysis/F_VN_CreateBandpassButterworthFilter

	{attribute 'TcIecLibraryType'}
	{attribute 'external_name' := 'F_VN_CreateBandpassButterworthFilter_GUID_BC7C26E5_AE80_D86F_AF9B_27858718E399'}
	(* Creates a bandpass Butterworth filter, which can be applied to a frequency domain image by element-wise multiplication. *)
	FUNCTION F_VN_CreateBandpassButterworthFilter : HRESULT
	VAR_INPUT
		ipFilter	:	REFERENCE TO ITcVnImage;	(* Returns the created filter (1 channel of type REAL or LREAL, depending on bDoublePrecision. Non-zero interface pointers are reused.). *)
		nWidth	:	UDINT;	(* Filter width (even, >= 2, must match the width of the image it is applied to) *)
		nHeight	:	UDINT;	(* Filter height (even, >= 2, must match the height of the image it is applied to) *)
		bDoublePrecision	:	BOOL;	(* If true, the filter is generated with double precision (LREAL) instead of single precision (REAL). *)
		bOriginAtCenter	:	BOOL;	(* If true, the filter origin is shifted to the image center. *)
		fCutoffDistance	:	LREAL;	(* The cutoff distance of the Butterworth filter (> 0). *)
		fBandWidth	:	LREAL;	(* The band width of the Butterworth filter (> 0). *)
		nOrder	:	UDINT;	(* The order of the Butterworth filter (> 0). *)
		fScale	:	LREAL;	(* The scale factor of the Butterworth filter denominator term (> 0, e.g. 0.414 or 1.0). *)
		hrPrev	:	HRESULT;	(* HRESULT indicating the result of previous operations (If SUCCEEDED(hrPrev) equals false, no operation is executed.) *)
	END_VAR

END_FUNCTION

// Functions/Fourier Analysis/F_VN_CreateBandpassGaussianFilter

	{attribute 'TcIecLibraryType'}
	{attribute 'external_name' := 'F_VN_CreateBandpassGaussianFilter_GUID_B333B228_9C73_DB11_9D49_31EC594A2466'}
	(* Creates a bandpass Gaussian filter, which can be applied to a frequency domain image by element-wise multiplication. *)
	FUNCTION F_VN_CreateBandpassGaussianFilter : HRESULT
	VAR_INPUT
		ipFilter	:	REFERENCE TO ITcVnImage;	(* Returns the created filter (1 channel of type REAL or LREAL, depending on bDoublePrecision. Non-zero interface pointers are reused.). *)
		nWidth	:	UDINT;	(* Filter width (even, >= 2, must match the width of the image it is applied to) *)
		nHeight	:	UDINT;	(* Filter height (even, >= 2, must match the height of the image it is applied to) *)
		bDoublePrecision	:	BOOL;	(* If true, the filter is generated with double precision (LREAL) instead of single precision (REAL). *)
		bOriginAtCenter	:	BOOL;	(* If true, the filter origin is shifted to the image center. *)
		fCutoffDistance	:	LREAL;	(* The cutoff distance of the Gaussian filter (> 0). *)
		fBandWidth	:	LREAL;	(* The band width of the Gaussian filter (> 0). *)
		hrPrev	:	HRESULT;	(* HRESULT indicating the result of previous operations (If SUCCEEDED(hrPrev) equals false, no operation is executed.) *)
	END_VAR

END_FUNCTION

// Functions/Fourier Analysis/F_VN_CreateBandrejectButterworthFilter

	{attribute 'TcIecLibraryType'}
	{attribute 'external_name' := 'F_VN_CreateBandrejectButterworthFilter_GUID_5BF0B1AD_04FB_D988_8353_BA8B3D56D2D8'}
	(* Creates a bandreject Butterworth filter, which can be applied to a frequency domain image by element-wise multiplication. *)
	FUNCTION F_VN_CreateBandrejectButterworthFilter : HRESULT
	VAR_INPUT
		ipFilter	:	REFERENCE TO ITcVnImage;	(* Returns the created filter (1 channel of type REAL or LREAL, depending on bDoublePrecision. Non-zero interface pointers are reused.). *)
		nWidth	:	UDINT;	(* Filter width (even, >= 2, must match the width of the image it is applied to) *)
		nHeight	:	UDINT;	(* Filter height (even, >= 2, must match the height of the image it is applied to) *)
		bDoublePrecision	:	BOOL;	(* If true, the filter is generated with double precision (LREAL) instead of single precision (REAL). *)
		bOriginAtCenter	:	BOOL;	(* If true, the filter origin is shifted to the image center. *)
		fCutoffDistance	:	LREAL;	(* The cutoff distance of the Butterworth filter (> 0). *)
		fBandWidth	:	LREAL;	(* The band width of the Butterworth filter (> 0). *)
		nOrder	:	UDINT;	(* The order of the Butterworth filter (> 0). *)
		fScale	:	LREAL;	(* The scale factor of the Butterworth filter denominator term (> 0, e.g. 0.414 or 1.0). *)
		hrPrev	:	HRESULT;	(* HRESULT indicating the result of previous operations (If SUCCEEDED(hrPrev) equals false, no operation is executed.) *)
	END_VAR

END_FUNCTION

// Functions/Fourier Analysis/F_VN_CreateBandrejectGaussianFilter

	{attribute 'TcIecLibraryType'}
	{attribute 'external_name' := 'F_VN_CreateBandrejectGaussianFilter_GUID_350EB3EA_FA46_DBB8_9331_FF0E9578B41B'}
	(* Creates a bandreject Gaussian filter, which can be applied to a frequency domain image by element-wise multiplication. *)
	FUNCTION F_VN_CreateBandrejectGaussianFilter : HRESULT
	VAR_INPUT
		ipFilter	:	REFERENCE TO ITcVnImage;	(* Returns the created filter (1 channel of type REAL or LREAL, depending on bDoublePrecision. Non-zero interface pointers are reused.). *)
		nWidth	:	UDINT;	(* Filter width (even, >= 2, must match the width of the image it is applied to) *)
		nHeight	:	UDINT;	(* Filter height (even, >= 2, must match the height of the image it is applied to) *)
		bDoublePrecision	:	BOOL;	(* If true, the filter is generated with double precision (LREAL) instead of single precision (REAL). *)
		bOriginAtCenter	:	BOOL;	(* If true, the filter origin is shifted to the image center. *)
		fCutoffDistance	:	LREAL;	(* The cutoff distance of the Gaussian filter (> 0). *)
		fBandWidth	:	LREAL;	(* The band width of the Gaussian filter (> 0). *)
		hrPrev	:	HRESULT;	(* HRESULT indicating the result of previous operations (If SUCCEEDED(hrPrev) equals false, no operation is executed.) *)
	END_VAR

END_FUNCTION

// Functions/Fourier Analysis/F_VN_CreateHighpassButterworthFilter

	{attribute 'TcIecLibraryType'}
	{attribute 'external_name' := 'F_VN_CreateHighpassButterworthFilter_GUID_3E3CE7D0_FAFF_D5EC_84AD_5750C9DB8770'}
	(* Creates a highpass Butterworth filter, which can be applied to a frequency domain image by element-wise multiplication. *)
	FUNCTION F_VN_CreateHighpassButterworthFilter : HRESULT
	VAR_INPUT
		ipFilter	:	REFERENCE TO ITcVnImage;	(* Returns the created filter (1 channel of type REAL or LREAL, depending on bDoublePrecision. Non-zero interface pointers are reused.). *)
		nWidth	:	UDINT;	(* Filter width (even, >= 2, must match the width of the image it is applied to) *)
		nHeight	:	UDINT;	(* Filter height (even, >= 2, must match the height of the image it is applied to) *)
		bDoublePrecision	:	BOOL;	(* If true, the filter is generated with double precision (LREAL) instead of single precision (REAL). *)
		bOriginAtCenter	:	BOOL;	(* If true, the filter origin is shifted to the image center. *)
		fCutoffDistance	:	LREAL;	(* The cutoff distance of the Butterworth filter (> 0). *)
		nOrder	:	UDINT;	(* The order of the Butterworth filter (> 0). *)
		fScale	:	LREAL;	(* The scale factor of the Butterworth filter denominator term (> 0, e.g. 0.414 or 1.0). *)
		hrPrev	:	HRESULT;	(* HRESULT indicating the result of previous operations (If SUCCEEDED(hrPrev) equals false, no operation is executed.) *)
	END_VAR

END_FUNCTION

// Functions/Fourier Analysis/F_VN_CreateHighpassGaussianFilter

